HMI tags "2080TN450A01Z02"
   "2080TN450A01Z02.MSW" : 52809b66-421d-457f-8884-6f7a49d4e247 AT %DB5129.DBX18.0, 500 ms
   "2080TN450A01Z02.DefaultText" : TextRef, internal   // Заголовок POPUP окна. При експорте из ECS через скрипт заполняется автоматически, если теги копируются в ручную то требуется в ручную задатать свойство Start Value
   "2080TN450A01Z02.BlockInfo" : Array [0..2] of Int AT %DB5129.DBX38.0, 500 ms
   "2080TN450A01Z02.StatusWork" : Int AT %DB5129.DBW242, 500 ms
   "2080TN450A01Z02.FP_PARAM.DampingTime" : Int AT %DB5129.DBW50, 500 ms
   "2080TN450A01Z02.FP_PARAM.Force_Value" : Real AT %DB5129.DBD52, 500 ms
   "2080TN450A01Z02.FP_PARAM.Scale_Min" : Real AT %DB5129.DBD56, 500 ms
   "2080TN450A01Z02.FP_PARAM.Scale_Max" : Real AT %DB5129.DBD60, 500 ms
   "2080TN450A01Z02.FP_PARAM.Gradient" : Real AT %DB5129.DBD64, 500 ms
   "2080TN450A01Z02.FP_PARAM.Grad_Pos" : Real AT %DB5129.DBD68, 500 ms
   "2080TN450A01Z02.FP_PARAM.Grad_Neg" : Real AT %DB5129.DBD72, 500 ms
   "2080TN450A01Z02.FP_PARAM.Grad_X" : Real AT %DB5129.DBD76, 500 ms
   "2080TN450A01Z02.FP_PARAM.Gradient_Time_Pre" : Int AT %DB5129.DBW80, 500 ms
   "2080TN450A01Z02.FP_PARAM.Gradient_Time_ACC" : Int AT %DB5129.DBW82, 500 ms
   "2080TN450A01Z02.FP_PARAM.Alarm_Hyst" : Real AT %DB5129.DBD84, 500 ms
   "2080TN450A01Z02.FP_PARAM.AlarmLimit_H3" : Real AT %DB5129.DBD88, 500 ms
   "2080TN450A01Z02.FP_PARAM.AlarmLimit_H2" : Real AT %DB5129.DBD92, 500 ms
   "2080TN450A01Z02.FP_PARAM.AlarmLimit_H1" : Real AT %DB5129.DBD96, 500 ms
   "2080TN450A01Z02.FP_PARAM.AlarmLimit_L1" : Real AT %DB5129.DBD100, 500 ms
   "2080TN450A01Z02.FP_PARAM.AlarmLimit_L2" : Real AT %DB5129.DBD104, 500 ms
   "2080TN450A01Z02.FP_PARAM.AlarmLimit_L3" : Real AT %DB5129.DBD108, 500 ms
   "2080TN450A01Z02.FP_PARAM.AlarmDelay_H3_Pre" : Int AT %DB5129.DBW112, 500 ms
   "2080TN450A01Z02.FP_PARAM.AlarmDelay_H3_Acc" : Int AT %DB5129.DBW114, 500 ms
   "2080TN450A01Z02.FP_PARAM.AlarmDelay_H2_Pre" : Int AT %DB5129.DBW116, 500 ms
   "2080TN450A01Z02.FP_PARAM.AlarmDelay_H2_Acc" : Int AT %DB5129.DBW118, 500 ms
   "2080TN450A01Z02.FP_PARAM.AlarmDelay_H1_Pre" : Int AT %DB5129.DBW120, 500 ms
   "2080TN450A01Z02.FP_PARAM.AlarmDelay_H1_Acc" : Int AT %DB5129.DBW122, 500 ms
   "2080TN450A01Z02.FP_PARAM.AlarmDelay_L1_Pre" : Int AT %DB5129.DBW124, 500 ms
   "2080TN450A01Z02.FP_PARAM.AlarmDelay_L1_Acc" : Int AT %DB5129.DBW126, 500 ms
   "2080TN450A01Z02.FP_PARAM.AlarmDelay_L2_Pre" : Int AT %DB5129.DBW128, 500 ms
   "2080TN450A01Z02.FP_PARAM.AlarmDelay_L2_Acc" : Int AT %DB5129.DBW130, 500 ms
   "2080TN450A01Z02.FP_PARAM.AlarmDelay_L3_Pre" : Int AT %DB5129.DBW132, 500 ms
   "2080TN450A01Z02.FP_PARAM.AlarmDelay_L3_Acc" : Int AT %DB5129.DBW134, 500 ms
   "2080TN450A01Z02.FP_PARAM.OpenLoopDelay_Pre" : Int AT %DB5129.DBW136, 500 ms
   "2080TN450A01Z02.FP_PARAM.OpenLoopDelay_Acc" : Int AT %DB5129.DBW138, 500 ms
   "2080TN450A01Z02.FP_PARAM.OverRangeDelay_Pre" : Int AT %DB5129.DBW140, 500 ms
   "2080TN450A01Z02.FP_PARAM.OverRangeDelay_Acc" : Int AT %DB5129.DBW142, 500 ms
   "2080TN450A01Z02.FP_PARAM.AuxLimit_H2_Value" : Real AT %DB5129.DBD144, 500 ms
   "2080TN450A01Z02.FP_PARAM.AuxLimit_H1_Value" : Real AT %DB5129.DBD148, 500 ms
   "2080TN450A01Z02.FP_PARAM.AuxLimit_L2_Value" : Real AT %DB5129.DBD152, 500 ms
   "2080TN450A01Z02.FP_PARAM.AuxLimit_L1_Value" : Real AT %DB5129.DBD156, 500 ms
   "2080TN450A01Z02.Unit" : TextRef, internal   // Еденицы измерения При експорте из ECS через скрипт заполняется автоматически, если теги копируются в ручную то требуется задатать свойство Text
   "2080TN450A01Z02.Decimals" : TextRef, internal   // Формат отображения При експорте из ECS через скрипт, заполняется автоматически. Если теги копируются в ручную то требуется задатать свойство Text s999999.9
   "2080TN450A01Z02.FP_EN.Square" : Bool AT %DB5129.DBX46.0, 500 ms
   "2080TN450A01Z02.FP_EN.SquareRoot" : Bool AT %DB5129.DBX46.1, 500 ms
   "2080TN450A01Z02.FP_EN.ParentSupress" : Bool AT %DB5129.DBX46.2, 500 ms
   "2080TN450A01Z02.FP_EN.ParentSupressUnit" : Bool AT %DB5129.DBX46.3, 500 ms
   "2080TN450A01Z02.FP_EN.Force" : Bool AT %DB5129.DBX46.4, 500 ms
   "2080TN450A01Z02.FP_EN.Damping" : Bool AT %DB5129.DBX46.5, 500 ms
   "2080TN450A01Z02.FP_EN.Gradient_Pos" : Bool AT %DB5129.DBX46.6, 500 ms
   "2080TN450A01Z02.FP_EN.Gradient_Neg" : Bool AT %DB5129.DBX46.7, 500 ms
   "2080TN450A01Z02.FP_EN.Hysteresis" : Bool AT %DB5129.DBX47.0, 500 ms
   "2080TN450A01Z02.FP_EN.Alarm_H3" : Bool AT %DB5129.DBX47.1, 500 ms
   "2080TN450A01Z02.FP_EN.Alarm_H2" : Bool AT %DB5129.DBX47.2, 500 ms
   "2080TN450A01Z02.FP_EN.Alarm_H1" : Bool AT %DB5129.DBX47.3, 500 ms
   "2080TN450A01Z02.FP_EN.Alarm_L1" : Bool AT %DB5129.DBX47.4, 500 ms
   "2080TN450A01Z02.FP_EN.Alarm_L2" : Bool AT %DB5129.DBX47.5, 500 ms
   "2080TN450A01Z02.FP_EN.Alarm_L3" : Bool AT %DB5129.DBX47.6, 500 ms
   "2080TN450A01Z02.FP_EN.AlarmDelay_H3" : Bool AT %DB5129.DBX47.7, 500 ms
   "2080TN450A01Z02.FP_EN.AlarmDelay_H2" : Bool AT %DB5129.DBX48.0, 500 ms
   "2080TN450A01Z02.FP_EN.AlarmDelay_H1" : Bool AT %DB5129.DBX48.1, 500 ms
   "2080TN450A01Z02.FP_EN.AlarmDelay_L1" : Bool AT %DB5129.DBX48.2, 500 ms
   "2080TN450A01Z02.FP_EN.AlarmDelay_L2" : Bool AT %DB5129.DBX48.3, 500 ms
   "2080TN450A01Z02.FP_EN.AlarmDelay_L3" : Bool AT %DB5129.DBX48.4, 500 ms
   "2080TN450A01Z02.FP_EN.ROC_Warn" : Bool AT %DB5129.DBX48.5, 500 ms
   "2080TN450A01Z02.FP_EN.U_Range_Warn" : Bool AT %DB5129.DBX48.6, 500 ms
   "2080TN450A01Z02.FP_EN.O_Range_Warn" : Bool AT %DB5129.DBX48.7, 500 ms
   "2080TN450A01Z02.trend_tag_name" : TextRef, internal   // Еденицы измерения При експорте из ECS через скрипт - заполняется автоматически, если теги копируются в ручную то требуется задатать свойство Text - имя тега для тренда
   "2080TN450A01Z02.DQ.AL_H3" : Bool AT %DB5129.DBX16.0, 500 ms
   "2080TN450A01Z02.DQ.AL_H2" : Bool AT %DB5129.DBX16.1, 500 ms
   "2080TN450A01Z02.DQ.AL_H1" : Bool AT %DB5129.DBX16.2, 500 ms
   "2080TN450A01Z02.DQ.AL_L1" : Bool AT %DB5129.DBX16.3, 500 ms
   "2080TN450A01Z02.DQ.AL_L2" : Bool AT %DB5129.DBX16.4, 500 ms
   "2080TN450A01Z02.DQ.AL_L3" : Bool AT %DB5129.DBX16.5, 500 ms
   "2080TN450A01Z02.DQ.SIG_OK" : Bool AT %DB5129.DBX16.6, 500 ms
   "2080TN450A01Z02.DQ.LIM_H2" : Bool AT %DB5129.DBX16.7, 500 ms
   "2080TN450A01Z02.DQ.LIM_H1" : Bool AT %DB5129.DBX17.0, 500 ms
   "2080TN450A01Z02.DQ.LIM_L1" : Bool AT %DB5129.DBX17.1, 500 ms
   "2080TN450A01Z02.DQ.LIM_L2" : Bool AT %DB5129.DBX17.2, 500 ms
   "2080TN450A01Z02.DQ.GR_P" : Bool AT %DB5129.DBX17.3, 500 ms
   "2080TN450A01Z02.DQ.GR_N" : Bool AT %DB5129.DBX17.4, 500 ms
   "2080TN450A01Z02.I.IN" : Real AT %DB5129.DBD2, 500 ms
   "2080TN450A01Z02.I.SIG_TYPE" : Int AT %DB5129.DBW0, 500 ms
   "2080TN450A01Z02.I.FI_BUS" : Byte AT %DB5129.DBB6, 500 ms
   "2080TN450A01Z02.DI.U_RANGE" : Bool AT %DB5129.DBX7.0, 500 ms
   "2080TN450A01Z02.DI.O_RANGE" : Bool AT %DB5129.DBX7.1, 500 ms
   "2080TN450A01Z02.DI.SIG_FAULT" : Bool AT %DB5129.DBX7.2, 500 ms
   "2080TN450A01Z02.DI.EnConfig" : Bool AT %DB5129.DBX7.3, 500 ms
   "2080TN450A01Z02.DI.AEN" : Bool AT %DB5129.DBX7.4, 500 ms
   "2080TN450A01Z02.DI.AL_SUPR" : Bool AT %DB5129.DBX7.5, 500 ms
   "2080TN450A01Z02.Q.PV_NORM" : Real AT %DB5129.DBD8, 500 ms
   "2080TN450A01Z02.Q.PV_SCAL" : Real AT %DB5129.DBD12, 500 ms
   "2080TN450A01Z02.ParentInfo" : TextRef, internal   // Имя родителя для попап окна, вкладка инфо. При експорте из ECS через скрипт заполняется автоматически, если теги копируются в ручную то требуется в ручную задатать свойство Start Value

HMI tags "2080TN450A01Z03"
   "2080TN450A01Z03.MSW" : 52809b66-421d-457f-8884-6f7a49d4e247 AT %DB5130.DBX18.0, 500 ms
   "2080TN450A01Z03.DefaultText" : TextRef, internal   // Заголовок POPUP окна. При експорте из ECS через скрипт заполняется автоматически, если теги копируются в ручную то требуется в ручную задатать свойство Start Value
   "2080TN450A01Z03.BlockInfo" : Array [0..2] of Int AT %DB5130.DBX38.0, 500 ms
   "2080TN450A01Z03.StatusWork" : Int AT %DB5130.DBW242, 500 ms
   "2080TN450A01Z03.FP_PARAM.DampingTime" : Int AT %DB5130.DBW50, 500 ms
   "2080TN450A01Z03.FP_PARAM.Force_Value" : Real AT %DB5130.DBD52, 500 ms
   "2080TN450A01Z03.FP_PARAM.Scale_Min" : Real AT %DB5130.DBD56, 500 ms
   "2080TN450A01Z03.FP_PARAM.Scale_Max" : Real AT %DB5130.DBD60, 500 ms
   "2080TN450A01Z03.FP_PARAM.Gradient" : Real AT %DB5130.DBD64, 500 ms
   "2080TN450A01Z03.FP_PARAM.Grad_Pos" : Real AT %DB5130.DBD68, 500 ms
   "2080TN450A01Z03.FP_PARAM.Grad_Neg" : Real AT %DB5130.DBD72, 500 ms
   "2080TN450A01Z03.FP_PARAM.Grad_X" : Real AT %DB5130.DBD76, 500 ms
   "2080TN450A01Z03.FP_PARAM.Gradient_Time_Pre" : Int AT %DB5130.DBW80, 500 ms
   "2080TN450A01Z03.FP_PARAM.Gradient_Time_ACC" : Int AT %DB5130.DBW82, 500 ms
   "2080TN450A01Z03.FP_PARAM.Alarm_Hyst" : Real AT %DB5130.DBD84, 500 ms
   "2080TN450A01Z03.FP_PARAM.AlarmLimit_H3" : Real AT %DB5130.DBD88, 500 ms
   "2080TN450A01Z03.FP_PARAM.AlarmLimit_H2" : Real AT %DB5130.DBD92, 500 ms
   "2080TN450A01Z03.FP_PARAM.AlarmLimit_H1" : Real AT %DB5130.DBD96, 500 ms
   "2080TN450A01Z03.FP_PARAM.AlarmLimit_L1" : Real AT %DB5130.DBD100, 500 ms
   "2080TN450A01Z03.FP_PARAM.AlarmLimit_L2" : Real AT %DB5130.DBD104, 500 ms
   "2080TN450A01Z03.FP_PARAM.AlarmLimit_L3" : Real AT %DB5130.DBD108, 500 ms
   "2080TN450A01Z03.FP_PARAM.AlarmDelay_H3_Pre" : Int AT %DB5130.DBW112, 500 ms
   "2080TN450A01Z03.FP_PARAM.AlarmDelay_H3_Acc" : Int AT %DB5130.DBW114, 500 ms
   "2080TN450A01Z03.FP_PARAM.AlarmDelay_H2_Pre" : Int AT %DB5130.DBW116, 500 ms
   "2080TN450A01Z03.FP_PARAM.AlarmDelay_H2_Acc" : Int AT %DB5130.DBW118, 500 ms
   "2080TN450A01Z03.FP_PARAM.AlarmDelay_H1_Pre" : Int AT %DB5130.DBW120, 500 ms
   "2080TN450A01Z03.FP_PARAM.AlarmDelay_H1_Acc" : Int AT %DB5130.DBW122, 500 ms
   "2080TN450A01Z03.FP_PARAM.AlarmDelay_L1_Pre" : Int AT %DB5130.DBW124, 500 ms
   "2080TN450A01Z03.FP_PARAM.AlarmDelay_L1_Acc" : Int AT %DB5130.DBW126, 500 ms
   "2080TN450A01Z03.FP_PARAM.AlarmDelay_L2_Pre" : Int AT %DB5130.DBW128, 500 ms
   "2080TN450A01Z03.FP_PARAM.AlarmDelay_L2_Acc" : Int AT %DB5130.DBW130, 500 ms
   "2080TN450A01Z03.FP_PARAM.AlarmDelay_L3_Pre" : Int AT %DB5130.DBW132, 500 ms
   "2080TN450A01Z03.FP_PARAM.AlarmDelay_L3_Acc" : Int AT %DB5130.DBW134, 500 ms
   "2080TN450A01Z03.FP_PARAM.OpenLoopDelay_Pre" : Int AT %DB5130.DBW136, 500 ms
   "2080TN450A01Z03.FP_PARAM.OpenLoopDelay_Acc" : Int AT %DB5130.DBW138, 500 ms
   "2080TN450A01Z03.FP_PARAM.OverRangeDelay_Pre" : Int AT %DB5130.DBW140, 500 ms
   "2080TN450A01Z03.FP_PARAM.OverRangeDelay_Acc" : Int AT %DB5130.DBW142, 500 ms
   "2080TN450A01Z03.FP_PARAM.AuxLimit_H2_Value" : Real AT %DB5130.DBD144, 500 ms
   "2080TN450A01Z03.FP_PARAM.AuxLimit_H1_Value" : Real AT %DB5130.DBD148, 500 ms
   "2080TN450A01Z03.FP_PARAM.AuxLimit_L2_Value" : Real AT %DB5130.DBD152, 500 ms
   "2080TN450A01Z03.FP_PARAM.AuxLimit_L1_Value" : Real AT %DB5130.DBD156, 500 ms
   "2080TN450A01Z03.Unit" : TextRef, internal   // Еденицы измерения При експорте из ECS через скрипт заполняется автоматически, если теги копируются в ручную то требуется задатать свойство Text
   "2080TN450A01Z03.Decimals" : TextRef, internal   // Формат отображения При експорте из ECS через скрипт, заполняется автоматически. Если теги копируются в ручную то требуется задатать свойство Text s999999.9
   "2080TN450A01Z03.FP_EN.Square" : Bool AT %DB5130.DBX46.0, 500 ms
   "2080TN450A01Z03.FP_EN.SquareRoot" : Bool AT %DB5130.DBX46.1, 500 ms
   "2080TN450A01Z03.FP_EN.ParentSupress" : Bool AT %DB5130.DBX46.2, 500 ms
   "2080TN450A01Z03.FP_EN.ParentSupressUnit" : Bool AT %DB5130.DBX46.3, 500 ms
   "2080TN450A01Z03.FP_EN.Force" : Bool AT %DB5130.DBX46.4, 500 ms
   "2080TN450A01Z03.FP_EN.Damping" : Bool AT %DB5130.DBX46.5, 500 ms
   "2080TN450A01Z03.FP_EN.Gradient_Pos" : Bool AT %DB5130.DBX46.6, 500 ms
   "2080TN450A01Z03.FP_EN.Gradient_Neg" : Bool AT %DB5130.DBX46.7, 500 ms
   "2080TN450A01Z03.FP_EN.Hysteresis" : Bool AT %DB5130.DBX47.0, 500 ms
   "2080TN450A01Z03.FP_EN.Alarm_H3" : Bool AT %DB5130.DBX47.1, 500 ms
   "2080TN450A01Z03.FP_EN.Alarm_H2" : Bool AT %DB5130.DBX47.2, 500 ms
   "2080TN450A01Z03.FP_EN.Alarm_H1" : Bool AT %DB5130.DBX47.3, 500 ms
   "2080TN450A01Z03.FP_EN.Alarm_L1" : Bool AT %DB5130.DBX47.4, 500 ms
   "2080TN450A01Z03.FP_EN.Alarm_L2" : Bool AT %DB5130.DBX47.5, 500 ms
   "2080TN450A01Z03.FP_EN.Alarm_L3" : Bool AT %DB5130.DBX47.6, 500 ms
   "2080TN450A01Z03.FP_EN.AlarmDelay_H3" : Bool AT %DB5130.DBX47.7, 500 ms
   "2080TN450A01Z03.FP_EN.AlarmDelay_H2" : Bool AT %DB5130.DBX48.0, 500 ms
   "2080TN450A01Z03.FP_EN.AlarmDelay_H1" : Bool AT %DB5130.DBX48.1, 500 ms
   "2080TN450A01Z03.FP_EN.AlarmDelay_L1" : Bool AT %DB5130.DBX48.2, 500 ms
   "2080TN450A01Z03.FP_EN.AlarmDelay_L2" : Bool AT %DB5130.DBX48.3, 500 ms
   "2080TN450A01Z03.FP_EN.AlarmDelay_L3" : Bool AT %DB5130.DBX48.4, 500 ms
   "2080TN450A01Z03.FP_EN.ROC_Warn" : Bool AT %DB5130.DBX48.5, 500 ms
   "2080TN450A01Z03.FP_EN.U_Range_Warn" : Bool AT %DB5130.DBX48.6, 500 ms
   "2080TN450A01Z03.FP_EN.O_Range_Warn" : Bool AT %DB5130.DBX48.7, 500 ms
   "2080TN450A01Z03.trend_tag_name" : TextRef, internal   // Еденицы измерения При експорте из ECS через скрипт - заполняется автоматически, если теги копируются в ручную то требуется задатать свойство Text - имя тега для тренда
   "2080TN450A01Z03.DQ.AL_H3" : Bool AT %DB5130.DBX16.0, 500 ms
   "2080TN450A01Z03.DQ.AL_H2" : Bool AT %DB5130.DBX16.1, 500 ms
   "2080TN450A01Z03.DQ.AL_H1" : Bool AT %DB5130.DBX16.2, 500 ms
   "2080TN450A01Z03.DQ.AL_L1" : Bool AT %DB5130.DBX16.3, 500 ms
   "2080TN450A01Z03.DQ.AL_L2" : Bool AT %DB5130.DBX16.4, 500 ms
   "2080TN450A01Z03.DQ.AL_L3" : Bool AT %DB5130.DBX16.5, 500 ms
   "2080TN450A01Z03.DQ.SIG_OK" : Bool AT %DB5130.DBX16.6, 500 ms
   "2080TN450A01Z03.DQ.LIM_H2" : Bool AT %DB5130.DBX16.7, 500 ms
   "2080TN450A01Z03.DQ.LIM_H1" : Bool AT %DB5130.DBX17.0, 500 ms
   "2080TN450A01Z03.DQ.LIM_L1" : Bool AT %DB5130.DBX17.1, 500 ms
   "2080TN450A01Z03.DQ.LIM_L2" : Bool AT %DB5130.DBX17.2, 500 ms
   "2080TN450A01Z03.DQ.GR_P" : Bool AT %DB5130.DBX17.3, 500 ms
   "2080TN450A01Z03.DQ.GR_N" : Bool AT %DB5130.DBX17.4, 500 ms
   "2080TN450A01Z03.I.IN" : Real AT %DB5130.DBD2, 500 ms
   "2080TN450A01Z03.I.SIG_TYPE" : Int AT %DB5130.DBW0, 500 ms
   "2080TN450A01Z03.I.FI_BUS" : Byte AT %DB5130.DBB6, 500 ms
   "2080TN450A01Z03.DI.U_RANGE" : Bool AT %DB5130.DBX7.0, 500 ms
   "2080TN450A01Z03.DI.O_RANGE" : Bool AT %DB5130.DBX7.1, 500 ms
   "2080TN450A01Z03.DI.SIG_FAULT" : Bool AT %DB5130.DBX7.2, 500 ms
   "2080TN450A01Z03.DI.EnConfig" : Bool AT %DB5130.DBX7.3, 500 ms
   "2080TN450A01Z03.DI.AEN" : Bool AT %DB5130.DBX7.4, 500 ms
   "2080TN450A01Z03.DI.AL_SUPR" : Bool AT %DB5130.DBX7.5, 500 ms
   "2080TN450A01Z03.Q.PV_NORM" : Real AT %DB5130.DBD8, 500 ms
   "2080TN450A01Z03.Q.PV_SCAL" : Real AT %DB5130.DBD12, 500 ms
   "2080TN450A01Z03.ParentInfo" : TextRef, internal   // Имя родителя для попап окна, вкладка инфо. При експорте из ECS через скрипт заполняется автоматически, если теги копируются в ручную то требуется в ручную задатать свойство Start Value

HMI tags "2080TN450A01Z05"
   "2080TN450A01Z05.MSW" : 52809b66-421d-457f-8884-6f7a49d4e247 AT %DB5139.DBX18.0, 500 ms
   "2080TN450A01Z05.DefaultText" : TextRef, internal   // Заголовок POPUP окна. При експорте из ECS через скрипт заполняется автоматически, если теги копируются в ручную то требуется в ручную задатать свойство Start Value
   "2080TN450A01Z05.BlockInfo" : Array [0..2] of Int AT %DB5139.DBX38.0, 500 ms
   "2080TN450A01Z05.StatusWork" : Int AT %DB5139.DBW242, 500 ms
   "2080TN450A01Z05.FP_PARAM.DampingTime" : Int AT %DB5139.DBW50, 500 ms
   "2080TN450A01Z05.FP_PARAM.Force_Value" : Real AT %DB5139.DBD52, 500 ms
   "2080TN450A01Z05.FP_PARAM.Scale_Min" : Real AT %DB5139.DBD56, 500 ms
   "2080TN450A01Z05.FP_PARAM.Scale_Max" : Real AT %DB5139.DBD60, 500 ms
   "2080TN450A01Z05.FP_PARAM.Gradient" : Real AT %DB5139.DBD64, 500 ms
   "2080TN450A01Z05.FP_PARAM.Grad_Pos" : Real AT %DB5139.DBD68, 500 ms
   "2080TN450A01Z05.FP_PARAM.Grad_Neg" : Real AT %DB5139.DBD72, 500 ms
   "2080TN450A01Z05.FP_PARAM.Grad_X" : Real AT %DB5139.DBD76, 500 ms
   "2080TN450A01Z05.FP_PARAM.Gradient_Time_Pre" : Int AT %DB5139.DBW80, 500 ms
   "2080TN450A01Z05.FP_PARAM.Gradient_Time_ACC" : Int AT %DB5139.DBW82, 500 ms
   "2080TN450A01Z05.FP_PARAM.Alarm_Hyst" : Real AT %DB5139.DBD84, 500 ms
   "2080TN450A01Z05.FP_PARAM.AlarmLimit_H3" : Real AT %DB5139.DBD88, 500 ms
   "2080TN450A01Z05.FP_PARAM.AlarmLimit_H2" : Real AT %DB5139.DBD92, 500 ms
   "2080TN450A01Z05.FP_PARAM.AlarmLimit_H1" : Real AT %DB5139.DBD96, 500 ms
   "2080TN450A01Z05.FP_PARAM.AlarmLimit_L1" : Real AT %DB5139.DBD100, 500 ms
   "2080TN450A01Z05.FP_PARAM.AlarmLimit_L2" : Real AT %DB5139.DBD104, 500 ms
   "2080TN450A01Z05.FP_PARAM.AlarmLimit_L3" : Real AT %DB5139.DBD108, 500 ms
   "2080TN450A01Z05.FP_PARAM.AlarmDelay_H3_Pre" : Int AT %DB5139.DBW112, 500 ms
   "2080TN450A01Z05.FP_PARAM.AlarmDelay_H3_Acc" : Int AT %DB5139.DBW114, 500 ms
   "2080TN450A01Z05.FP_PARAM.AlarmDelay_H2_Pre" : Int AT %DB5139.DBW116, 500 ms
   "2080TN450A01Z05.FP_PARAM.AlarmDelay_H2_Acc" : Int AT %DB5139.DBW118, 500 ms
   "2080TN450A01Z05.FP_PARAM.AlarmDelay_H1_Pre" : Int AT %DB5139.DBW120, 500 ms
   "2080TN450A01Z05.FP_PARAM.AlarmDelay_H1_Acc" : Int AT %DB5139.DBW122, 500 ms
   "2080TN450A01Z05.FP_PARAM.AlarmDelay_L1_Pre" : Int AT %DB5139.DBW124, 500 ms
   "2080TN450A01Z05.FP_PARAM.AlarmDelay_L1_Acc" : Int AT %DB5139.DBW126, 500 ms
   "2080TN450A01Z05.FP_PARAM.AlarmDelay_L2_Pre" : Int AT %DB5139.DBW128, 500 ms
   "2080TN450A01Z05.FP_PARAM.AlarmDelay_L2_Acc" : Int AT %DB5139.DBW130, 500 ms
   "2080TN450A01Z05.FP_PARAM.AlarmDelay_L3_Pre" : Int AT %DB5139.DBW132, 500 ms
   "2080TN450A01Z05.FP_PARAM.AlarmDelay_L3_Acc" : Int AT %DB5139.DBW134, 500 ms
   "2080TN450A01Z05.FP_PARAM.OpenLoopDelay_Pre" : Int AT %DB5139.DBW136, 500 ms
   "2080TN450A01Z05.FP_PARAM.OpenLoopDelay_Acc" : Int AT %DB5139.DBW138, 500 ms
   "2080TN450A01Z05.FP_PARAM.OverRangeDelay_Pre" : Int AT %DB5139.DBW140, 500 ms
   "2080TN450A01Z05.FP_PARAM.OverRangeDelay_Acc" : Int AT %DB5139.DBW142, 500 ms
   "2080TN450A01Z05.FP_PARAM.AuxLimit_H2_Value" : Real AT %DB5139.DBD144, 500 ms
   "2080TN450A01Z05.FP_PARAM.AuxLimit_H1_Value" : Real AT %DB5139.DBD148, 500 ms
   "2080TN450A01Z05.FP_PARAM.AuxLimit_L2_Value" : Real AT %DB5139.DBD152, 500 ms
   "2080TN450A01Z05.FP_PARAM.AuxLimit_L1_Value" : Real AT %DB5139.DBD156, 500 ms
   "2080TN450A01Z05.Unit" : TextRef, internal   // Еденицы измерения При експорте из ECS через скрипт заполняется автоматически, если теги копируются в ручную то требуется задатать свойство Text
   "2080TN450A01Z05.Decimals" : TextRef, internal   // Формат отображения При експорте из ECS через скрипт, заполняется автоматически. Если теги копируются в ручную то требуется задатать свойство Text s999999.9
   "2080TN450A01Z05.FP_EN.Square" : Bool AT %DB5139.DBX46.0, 500 ms
   "2080TN450A01Z05.FP_EN.SquareRoot" : Bool AT %DB5139.DBX46.1, 500 ms
   "2080TN450A01Z05.FP_EN.ParentSupress" : Bool AT %DB5139.DBX46.2, 500 ms
   "2080TN450A01Z05.FP_EN.ParentSupressUnit" : Bool AT %DB5139.DBX46.3, 500 ms
   "2080TN450A01Z05.FP_EN.Force" : Bool AT %DB5139.DBX46.4, 500 ms
   "2080TN450A01Z05.FP_EN.Damping" : Bool AT %DB5139.DBX46.5, 500 ms
   "2080TN450A01Z05.FP_EN.Gradient_Pos" : Bool AT %DB5139.DBX46.6, 500 ms
   "2080TN450A01Z05.FP_EN.Gradient_Neg" : Bool AT %DB5139.DBX46.7, 500 ms
   "2080TN450A01Z05.FP_EN.Hysteresis" : Bool AT %DB5139.DBX47.0, 500 ms
   "2080TN450A01Z05.FP_EN.Alarm_H3" : Bool AT %DB5139.DBX47.1, 500 ms
   "2080TN450A01Z05.FP_EN.Alarm_H2" : Bool AT %DB5139.DBX47.2, 500 ms
   "2080TN450A01Z05.FP_EN.Alarm_H1" : Bool AT %DB5139.DBX47.3, 500 ms
   "2080TN450A01Z05.FP_EN.Alarm_L1" : Bool AT %DB5139.DBX47.4, 500 ms
   "2080TN450A01Z05.FP_EN.Alarm_L2" : Bool AT %DB5139.DBX47.5, 500 ms
   "2080TN450A01Z05.FP_EN.Alarm_L3" : Bool AT %DB5139.DBX47.6, 500 ms
   "2080TN450A01Z05.FP_EN.AlarmDelay_H3" : Bool AT %DB5139.DBX47.7, 500 ms
   "2080TN450A01Z05.FP_EN.AlarmDelay_H2" : Bool AT %DB5139.DBX48.0, 500 ms
   "2080TN450A01Z05.FP_EN.AlarmDelay_H1" : Bool AT %DB5139.DBX48.1, 500 ms
   "2080TN450A01Z05.FP_EN.AlarmDelay_L1" : Bool AT %DB5139.DBX48.2, 500 ms
   "2080TN450A01Z05.FP_EN.AlarmDelay_L2" : Bool AT %DB5139.DBX48.3, 500 ms
   "2080TN450A01Z05.FP_EN.AlarmDelay_L3" : Bool AT %DB5139.DBX48.4, 500 ms
   "2080TN450A01Z05.FP_EN.ROC_Warn" : Bool AT %DB5139.DBX48.5, 500 ms
   "2080TN450A01Z05.FP_EN.U_Range_Warn" : Bool AT %DB5139.DBX48.6, 500 ms
   "2080TN450A01Z05.FP_EN.O_Range_Warn" : Bool AT %DB5139.DBX48.7, 500 ms
   "2080TN450A01Z05.trend_tag_name" : TextRef, internal   // Еденицы измерения При експорте из ECS через скрипт - заполняется автоматически, если теги копируются в ручную то требуется задатать свойство Text - имя тега для тренда
   "2080TN450A01Z05.DQ.AL_H3" : Bool AT %DB5139.DBX16.0, 500 ms
   "2080TN450A01Z05.DQ.AL_H2" : Bool AT %DB5139.DBX16.1, 500 ms
   "2080TN450A01Z05.DQ.AL_H1" : Bool AT %DB5139.DBX16.2, 500 ms
   "2080TN450A01Z05.DQ.AL_L1" : Bool AT %DB5139.DBX16.3, 500 ms
   "2080TN450A01Z05.DQ.AL_L2" : Bool AT %DB5139.DBX16.4, 500 ms
   "2080TN450A01Z05.DQ.AL_L3" : Bool AT %DB5139.DBX16.5, 500 ms
   "2080TN450A01Z05.DQ.SIG_OK" : Bool AT %DB5139.DBX16.6, 500 ms
   "2080TN450A01Z05.DQ.LIM_H2" : Bool AT %DB5139.DBX16.7, 500 ms
   "2080TN450A01Z05.DQ.LIM_H1" : Bool AT %DB5139.DBX17.0, 500 ms
   "2080TN450A01Z05.DQ.LIM_L1" : Bool AT %DB5139.DBX17.1, 500 ms
   "2080TN450A01Z05.DQ.LIM_L2" : Bool AT %DB5139.DBX17.2, 500 ms
   "2080TN450A01Z05.DQ.GR_P" : Bool AT %DB5139.DBX17.3, 500 ms
   "2080TN450A01Z05.DQ.GR_N" : Bool AT %DB5139.DBX17.4, 500 ms
   "2080TN450A01Z05.I.IN" : Real AT %DB5139.DBD2, 500 ms
   "2080TN450A01Z05.I.SIG_TYPE" : Int AT %DB5139.DBW0, 500 ms
   "2080TN450A01Z05.I.FI_BUS" : Byte AT %DB5139.DBB6, 500 ms
   "2080TN450A01Z05.DI.U_RANGE" : Bool AT %DB5139.DBX7.0, 500 ms
   "2080TN450A01Z05.DI.O_RANGE" : Bool AT %DB5139.DBX7.1, 500 ms
   "2080TN450A01Z05.DI.SIG_FAULT" : Bool AT %DB5139.DBX7.2, 500 ms
   "2080TN450A01Z05.DI.EnConfig" : Bool AT %DB5139.DBX7.3, 500 ms
   "2080TN450A01Z05.DI.AEN" : Bool AT %DB5139.DBX7.4, 500 ms
   "2080TN450A01Z05.DI.AL_SUPR" : Bool AT %DB5139.DBX7.5, 500 ms
   "2080TN450A01Z05.Q.PV_NORM" : Real AT %DB5139.DBD8, 500 ms
   "2080TN450A01Z05.Q.PV_SCAL" : Real AT %DB5139.DBD12, 500 ms
   "2080TN450A01Z05.ParentInfo" : TextRef, internal   // Имя родителя для попап окна, вкладка инфо. При експорте из ECS через скрипт заполняется автоматически, если теги копируются в ручную то требуется в ручную задатать свойство Start Value

HMI tags "2080TN450N01A01"
   "2080TN450N01A01.MSW" : 52809b66-421d-457f-8884-6f7a49d4e247 AT %DB5135.DBX18.0, 500 ms
   "2080TN450N01A01.DefaultText" : TextRef, internal   // Заголовок POPUP окна. При експорте из ECS через скрипт заполняется автоматически, если теги копируются в ручную то требуется в ручную задатать свойство Start Value
   "2080TN450N01A01.BlockInfo" : Array [0..2] of Int AT %DB5135.DBX38.0, 500 ms
   "2080TN450N01A01.StatusWork" : Int AT %DB5135.DBW242, 500 ms
   "2080TN450N01A01.FP_PARAM.DampingTime" : Int AT %DB5135.DBW50, 500 ms
   "2080TN450N01A01.FP_PARAM.Force_Value" : Real AT %DB5135.DBD52, 500 ms
   "2080TN450N01A01.FP_PARAM.Scale_Min" : Real AT %DB5135.DBD56, 500 ms
   "2080TN450N01A01.FP_PARAM.Scale_Max" : Real AT %DB5135.DBD60, 500 ms
   "2080TN450N01A01.FP_PARAM.Gradient" : Real AT %DB5135.DBD64, 500 ms
   "2080TN450N01A01.FP_PARAM.Grad_Pos" : Real AT %DB5135.DBD68, 500 ms
   "2080TN450N01A01.FP_PARAM.Grad_Neg" : Real AT %DB5135.DBD72, 500 ms
   "2080TN450N01A01.FP_PARAM.Grad_X" : Real AT %DB5135.DBD76, 500 ms
   "2080TN450N01A01.FP_PARAM.Gradient_Time_Pre" : Int AT %DB5135.DBW80, 500 ms
   "2080TN450N01A01.FP_PARAM.Gradient_Time_ACC" : Int AT %DB5135.DBW82, 500 ms
   "2080TN450N01A01.FP_PARAM.Alarm_Hyst" : Real AT %DB5135.DBD84, 500 ms
   "2080TN450N01A01.FP_PARAM.AlarmLimit_H3" : Real AT %DB5135.DBD88, 500 ms
   "2080TN450N01A01.FP_PARAM.AlarmLimit_H2" : Real AT %DB5135.DBD92, 500 ms
   "2080TN450N01A01.FP_PARAM.AlarmLimit_H1" : Real AT %DB5135.DBD96, 500 ms
   "2080TN450N01A01.FP_PARAM.AlarmLimit_L1" : Real AT %DB5135.DBD100, 500 ms
   "2080TN450N01A01.FP_PARAM.AlarmLimit_L2" : Real AT %DB5135.DBD104, 500 ms
   "2080TN450N01A01.FP_PARAM.AlarmLimit_L3" : Real AT %DB5135.DBD108, 500 ms
   "2080TN450N01A01.FP_PARAM.AlarmDelay_H3_Pre" : Int AT %DB5135.DBW112, 500 ms
   "2080TN450N01A01.FP_PARAM.AlarmDelay_H3_Acc" : Int AT %DB5135.DBW114, 500 ms
   "2080TN450N01A01.FP_PARAM.AlarmDelay_H2_Pre" : Int AT %DB5135.DBW116, 500 ms
   "2080TN450N01A01.FP_PARAM.AlarmDelay_H2_Acc" : Int AT %DB5135.DBW118, 500 ms
   "2080TN450N01A01.FP_PARAM.AlarmDelay_H1_Pre" : Int AT %DB5135.DBW120, 500 ms
   "2080TN450N01A01.FP_PARAM.AlarmDelay_H1_Acc" : Int AT %DB5135.DBW122, 500 ms
   "2080TN450N01A01.FP_PARAM.AlarmDelay_L1_Pre" : Int AT %DB5135.DBW124, 500 ms
   "2080TN450N01A01.FP_PARAM.AlarmDelay_L1_Acc" : Int AT %DB5135.DBW126, 500 ms
   "2080TN450N01A01.FP_PARAM.AlarmDelay_L2_Pre" : Int AT %DB5135.DBW128, 500 ms
   "2080TN450N01A01.FP_PARAM.AlarmDelay_L2_Acc" : Int AT %DB5135.DBW130, 500 ms
   "2080TN450N01A01.FP_PARAM.AlarmDelay_L3_Pre" : Int AT %DB5135.DBW132, 500 ms
   "2080TN450N01A01.FP_PARAM.AlarmDelay_L3_Acc" : Int AT %DB5135.DBW134, 500 ms
   "2080TN450N01A01.FP_PARAM.OpenLoopDelay_Pre" : Int AT %DB5135.DBW136, 500 ms
   "2080TN450N01A01.FP_PARAM.OpenLoopDelay_Acc" : Int AT %DB5135.DBW138, 500 ms
   "2080TN450N01A01.FP_PARAM.OverRangeDelay_Pre" : Int AT %DB5135.DBW140, 500 ms
   "2080TN450N01A01.FP_PARAM.OverRangeDelay_Acc" : Int AT %DB5135.DBW142, 500 ms
   "2080TN450N01A01.FP_PARAM.AuxLimit_H2_Value" : Real AT %DB5135.DBD144, 500 ms
   "2080TN450N01A01.FP_PARAM.AuxLimit_H1_Value" : Real AT %DB5135.DBD148, 500 ms
   "2080TN450N01A01.FP_PARAM.AuxLimit_L2_Value" : Real AT %DB5135.DBD152, 500 ms
   "2080TN450N01A01.FP_PARAM.AuxLimit_L1_Value" : Real AT %DB5135.DBD156, 500 ms
   "2080TN450N01A01.Unit" : TextRef, internal   // Еденицы измерения При експорте из ECS через скрипт заполняется автоматически, если теги копируются в ручную то требуется задатать свойство Text
   "2080TN450N01A01.Decimals" : TextRef, internal   // Формат отображения При експорте из ECS через скрипт, заполняется автоматически. Если теги копируются в ручную то требуется задатать свойство Text s999999.9
   "2080TN450N01A01.FP_EN.Square" : Bool AT %DB5135.DBX46.0, 500 ms
   "2080TN450N01A01.FP_EN.SquareRoot" : Bool AT %DB5135.DBX46.1, 500 ms
   "2080TN450N01A01.FP_EN.ParentSupress" : Bool AT %DB5135.DBX46.2, 500 ms
   "2080TN450N01A01.FP_EN.ParentSupressUnit" : Bool AT %DB5135.DBX46.3, 500 ms
   "2080TN450N01A01.FP_EN.Force" : Bool AT %DB5135.DBX46.4, 500 ms
   "2080TN450N01A01.FP_EN.Damping" : Bool AT %DB5135.DBX46.5, 500 ms
   "2080TN450N01A01.FP_EN.Gradient_Pos" : Bool AT %DB5135.DBX46.6, 500 ms
   "2080TN450N01A01.FP_EN.Gradient_Neg" : Bool AT %DB5135.DBX46.7, 500 ms
   "2080TN450N01A01.FP_EN.Hysteresis" : Bool AT %DB5135.DBX47.0, 500 ms
   "2080TN450N01A01.FP_EN.Alarm_H3" : Bool AT %DB5135.DBX47.1, 500 ms
   "2080TN450N01A01.FP_EN.Alarm_H2" : Bool AT %DB5135.DBX47.2, 500 ms
   "2080TN450N01A01.FP_EN.Alarm_H1" : Bool AT %DB5135.DBX47.3, 500 ms
   "2080TN450N01A01.FP_EN.Alarm_L1" : Bool AT %DB5135.DBX47.4, 500 ms
   "2080TN450N01A01.FP_EN.Alarm_L2" : Bool AT %DB5135.DBX47.5, 500 ms
   "2080TN450N01A01.FP_EN.Alarm_L3" : Bool AT %DB5135.DBX47.6, 500 ms
   "2080TN450N01A01.FP_EN.AlarmDelay_H3" : Bool AT %DB5135.DBX47.7, 500 ms
   "2080TN450N01A01.FP_EN.AlarmDelay_H2" : Bool AT %DB5135.DBX48.0, 500 ms
   "2080TN450N01A01.FP_EN.AlarmDelay_H1" : Bool AT %DB5135.DBX48.1, 500 ms
   "2080TN450N01A01.FP_EN.AlarmDelay_L1" : Bool AT %DB5135.DBX48.2, 500 ms
   "2080TN450N01A01.FP_EN.AlarmDelay_L2" : Bool AT %DB5135.DBX48.3, 500 ms
   "2080TN450N01A01.FP_EN.AlarmDelay_L3" : Bool AT %DB5135.DBX48.4, 500 ms
   "2080TN450N01A01.FP_EN.ROC_Warn" : Bool AT %DB5135.DBX48.5, 500 ms
   "2080TN450N01A01.FP_EN.U_Range_Warn" : Bool AT %DB5135.DBX48.6, 500 ms
   "2080TN450N01A01.FP_EN.O_Range_Warn" : Bool AT %DB5135.DBX48.7, 500 ms
   "2080TN450N01A01.trend_tag_name" : TextRef, internal   // Еденицы измерения При експорте из ECS через скрипт - заполняется автоматически, если теги копируются в ручную то требуется задатать свойство Text - имя тега для тренда
   "2080TN450N01A01.DQ.AL_H3" : Bool AT %DB5135.DBX16.0, 500 ms
   "2080TN450N01A01.DQ.AL_H2" : Bool AT %DB5135.DBX16.1, 500 ms
   "2080TN450N01A01.DQ.AL_H1" : Bool AT %DB5135.DBX16.2, 500 ms
   "2080TN450N01A01.DQ.AL_L1" : Bool AT %DB5135.DBX16.3, 500 ms
   "2080TN450N01A01.DQ.AL_L2" : Bool AT %DB5135.DBX16.4, 500 ms
   "2080TN450N01A01.DQ.AL_L3" : Bool AT %DB5135.DBX16.5, 500 ms
   "2080TN450N01A01.DQ.SIG_OK" : Bool AT %DB5135.DBX16.6, 500 ms
   "2080TN450N01A01.DQ.LIM_H2" : Bool AT %DB5135.DBX16.7, 500 ms
   "2080TN450N01A01.DQ.LIM_H1" : Bool AT %DB5135.DBX17.0, 500 ms
   "2080TN450N01A01.DQ.LIM_L1" : Bool AT %DB5135.DBX17.1, 500 ms
   "2080TN450N01A01.DQ.LIM_L2" : Bool AT %DB5135.DBX17.2, 500 ms
   "2080TN450N01A01.DQ.GR_P" : Bool AT %DB5135.DBX17.3, 500 ms
   "2080TN450N01A01.DQ.GR_N" : Bool AT %DB5135.DBX17.4, 500 ms
   "2080TN450N01A01.I.IN" : Real AT %DB5135.DBD2, 500 ms
   "2080TN450N01A01.I.SIG_TYPE" : Int AT %DB5135.DBW0, 500 ms
   "2080TN450N01A01.I.FI_BUS" : Byte AT %DB5135.DBB6, 500 ms
   "2080TN450N01A01.DI.U_RANGE" : Bool AT %DB5135.DBX7.0, 500 ms
   "2080TN450N01A01.DI.O_RANGE" : Bool AT %DB5135.DBX7.1, 500 ms
   "2080TN450N01A01.DI.SIG_FAULT" : Bool AT %DB5135.DBX7.2, 500 ms
   "2080TN450N01A01.DI.EnConfig" : Bool AT %DB5135.DBX7.3, 500 ms
   "2080TN450N01A01.DI.AEN" : Bool AT %DB5135.DBX7.4, 500 ms
   "2080TN450N01A01.DI.AL_SUPR" : Bool AT %DB5135.DBX7.5, 500 ms
   "2080TN450N01A01.Q.PV_NORM" : Real AT %DB5135.DBD8, 500 ms
   "2080TN450N01A01.Q.PV_SCAL" : Real AT %DB5135.DBD12, 500 ms
   "2080TN450N01A01.ParentInfo" : TextRef, internal   // Имя родителя для попап окна, вкладка инфо. При експорте из ECS через скрипт заполняется автоматически, если теги копируются в ручную то требуется в ручную задатать свойство Start Value

HMI tags "2080TN450N01I02"
   "2080TN450N01I02.MSW" : 52809b66-421d-457f-8884-6f7a49d4e247 AT %DB5112.DBX18.0, 500 ms
   "2080TN450N01I02.DefaultText" : TextRef, internal   // Заголовок POPUP окна. При експорте из ECS через скрипт заполняется автоматически, если теги копируются в ручную то требуется в ручную задатать свойство Start Value
   "2080TN450N01I02.BlockInfo" : Array [0..2] of Int AT %DB5112.DBX38.0, 500 ms
   "2080TN450N01I02.StatusWork" : Int AT %DB5112.DBW242, 500 ms
   "2080TN450N01I02.FP_PARAM.DampingTime" : Int AT %DB5112.DBW50, 500 ms
   "2080TN450N01I02.FP_PARAM.Force_Value" : Real AT %DB5112.DBD52, 500 ms
   "2080TN450N01I02.FP_PARAM.Scale_Min" : Real AT %DB5112.DBD56, 500 ms
   "2080TN450N01I02.FP_PARAM.Scale_Max" : Real AT %DB5112.DBD60, 500 ms
   "2080TN450N01I02.FP_PARAM.Gradient" : Real AT %DB5112.DBD64, 500 ms
   "2080TN450N01I02.FP_PARAM.Grad_Pos" : Real AT %DB5112.DBD68, 500 ms
   "2080TN450N01I02.FP_PARAM.Grad_Neg" : Real AT %DB5112.DBD72, 500 ms
   "2080TN450N01I02.FP_PARAM.Grad_X" : Real AT %DB5112.DBD76, 500 ms
   "2080TN450N01I02.FP_PARAM.Gradient_Time_Pre" : Int AT %DB5112.DBW80, 500 ms
   "2080TN450N01I02.FP_PARAM.Gradient_Time_ACC" : Int AT %DB5112.DBW82, 500 ms
   "2080TN450N01I02.FP_PARAM.Alarm_Hyst" : Real AT %DB5112.DBD84, 500 ms
   "2080TN450N01I02.FP_PARAM.AlarmLimit_H3" : Real AT %DB5112.DBD88, 500 ms
   "2080TN450N01I02.FP_PARAM.AlarmLimit_H2" : Real AT %DB5112.DBD92, 500 ms
   "2080TN450N01I02.FP_PARAM.AlarmLimit_H1" : Real AT %DB5112.DBD96, 500 ms
   "2080TN450N01I02.FP_PARAM.AlarmLimit_L1" : Real AT %DB5112.DBD100, 500 ms
   "2080TN450N01I02.FP_PARAM.AlarmLimit_L2" : Real AT %DB5112.DBD104, 500 ms
   "2080TN450N01I02.FP_PARAM.AlarmLimit_L3" : Real AT %DB5112.DBD108, 500 ms
   "2080TN450N01I02.FP_PARAM.AlarmDelay_H3_Pre" : Int AT %DB5112.DBW112, 500 ms
   "2080TN450N01I02.FP_PARAM.AlarmDelay_H3_Acc" : Int AT %DB5112.DBW114, 500 ms
   "2080TN450N01I02.FP_PARAM.AlarmDelay_H2_Pre" : Int AT %DB5112.DBW116, 500 ms
   "2080TN450N01I02.FP_PARAM.AlarmDelay_H2_Acc" : Int AT %DB5112.DBW118, 500 ms
   "2080TN450N01I02.FP_PARAM.AlarmDelay_H1_Pre" : Int AT %DB5112.DBW120, 500 ms
   "2080TN450N01I02.FP_PARAM.AlarmDelay_H1_Acc" : Int AT %DB5112.DBW122, 500 ms
   "2080TN450N01I02.FP_PARAM.AlarmDelay_L1_Pre" : Int AT %DB5112.DBW124, 500 ms
   "2080TN450N01I02.FP_PARAM.AlarmDelay_L1_Acc" : Int AT %DB5112.DBW126, 500 ms
   "2080TN450N01I02.FP_PARAM.AlarmDelay_L2_Pre" : Int AT %DB5112.DBW128, 500 ms
   "2080TN450N01I02.FP_PARAM.AlarmDelay_L2_Acc" : Int AT %DB5112.DBW130, 500 ms
   "2080TN450N01I02.FP_PARAM.AlarmDelay_L3_Pre" : Int AT %DB5112.DBW132, 500 ms
   "2080TN450N01I02.FP_PARAM.AlarmDelay_L3_Acc" : Int AT %DB5112.DBW134, 500 ms
   "2080TN450N01I02.FP_PARAM.OpenLoopDelay_Pre" : Int AT %DB5112.DBW136, 500 ms
   "2080TN450N01I02.FP_PARAM.OpenLoopDelay_Acc" : Int AT %DB5112.DBW138, 500 ms
   "2080TN450N01I02.FP_PARAM.OverRangeDelay_Pre" : Int AT %DB5112.DBW140, 500 ms
   "2080TN450N01I02.FP_PARAM.OverRangeDelay_Acc" : Int AT %DB5112.DBW142, 500 ms
   "2080TN450N01I02.FP_PARAM.AuxLimit_H2_Value" : Real AT %DB5112.DBD144, 500 ms
   "2080TN450N01I02.FP_PARAM.AuxLimit_H1_Value" : Real AT %DB5112.DBD148, 500 ms
   "2080TN450N01I02.FP_PARAM.AuxLimit_L2_Value" : Real AT %DB5112.DBD152, 500 ms
   "2080TN450N01I02.FP_PARAM.AuxLimit_L1_Value" : Real AT %DB5112.DBD156, 500 ms
   "2080TN450N01I02.Unit" : TextRef, internal   // Еденицы измерения При експорте из ECS через скрипт заполняется автоматически, если теги копируются в ручную то требуется задатать свойство Text
   "2080TN450N01I02.Decimals" : TextRef, internal   // Формат отображения При експорте из ECS через скрипт, заполняется автоматически. Если теги копируются в ручную то требуется задатать свойство Text s999999.9
   "2080TN450N01I02.FP_EN.Square" : Bool AT %DB5112.DBX46.0, 500 ms
   "2080TN450N01I02.FP_EN.SquareRoot" : Bool AT %DB5112.DBX46.1, 500 ms
   "2080TN450N01I02.FP_EN.ParentSupress" : Bool AT %DB5112.DBX46.2, 500 ms
   "2080TN450N01I02.FP_EN.ParentSupressUnit" : Bool AT %DB5112.DBX46.3, 500 ms
   "2080TN450N01I02.FP_EN.Force" : Bool AT %DB5112.DBX46.4, 500 ms
   "2080TN450N01I02.FP_EN.Damping" : Bool AT %DB5112.DBX46.5, 500 ms
   "2080TN450N01I02.FP_EN.Gradient_Pos" : Bool AT %DB5112.DBX46.6, 500 ms
   "2080TN450N01I02.FP_EN.Gradient_Neg" : Bool AT %DB5112.DBX46.7, 500 ms
   "2080TN450N01I02.FP_EN.Hysteresis" : Bool AT %DB5112.DBX47.0, 500 ms
   "2080TN450N01I02.FP_EN.Alarm_H3" : Bool AT %DB5112.DBX47.1, 500 ms
   "2080TN450N01I02.FP_EN.Alarm_H2" : Bool AT %DB5112.DBX47.2, 500 ms
   "2080TN450N01I02.FP_EN.Alarm_H1" : Bool AT %DB5112.DBX47.3, 500 ms
   "2080TN450N01I02.FP_EN.Alarm_L1" : Bool AT %DB5112.DBX47.4, 500 ms
   "2080TN450N01I02.FP_EN.Alarm_L2" : Bool AT %DB5112.DBX47.5, 500 ms
   "2080TN450N01I02.FP_EN.Alarm_L3" : Bool AT %DB5112.DBX47.6, 500 ms
   "2080TN450N01I02.FP_EN.AlarmDelay_H3" : Bool AT %DB5112.DBX47.7, 500 ms
   "2080TN450N01I02.FP_EN.AlarmDelay_H2" : Bool AT %DB5112.DBX48.0, 500 ms
   "2080TN450N01I02.FP_EN.AlarmDelay_H1" : Bool AT %DB5112.DBX48.1, 500 ms
   "2080TN450N01I02.FP_EN.AlarmDelay_L1" : Bool AT %DB5112.DBX48.2, 500 ms
   "2080TN450N01I02.FP_EN.AlarmDelay_L2" : Bool AT %DB5112.DBX48.3, 500 ms
   "2080TN450N01I02.FP_EN.AlarmDelay_L3" : Bool AT %DB5112.DBX48.4, 500 ms
   "2080TN450N01I02.FP_EN.ROC_Warn" : Bool AT %DB5112.DBX48.5, 500 ms
   "2080TN450N01I02.FP_EN.U_Range_Warn" : Bool AT %DB5112.DBX48.6, 500 ms
   "2080TN450N01I02.FP_EN.O_Range_Warn" : Bool AT %DB5112.DBX48.7, 500 ms
   "2080TN450N01I02.trend_tag_name" : TextRef, internal   // Еденицы измерения При експорте из ECS через скрипт - заполняется автоматически, если теги копируются в ручную то требуется задатать свойство Text - имя тега для тренда
   "2080TN450N01I02.DQ.AL_H3" : Bool AT %DB5112.DBX16.0, 500 ms
   "2080TN450N01I02.DQ.AL_H2" : Bool AT %DB5112.DBX16.1, 500 ms
   "2080TN450N01I02.DQ.AL_H1" : Bool AT %DB5112.DBX16.2, 500 ms
   "2080TN450N01I02.DQ.AL_L1" : Bool AT %DB5112.DBX16.3, 500 ms
   "2080TN450N01I02.DQ.AL_L2" : Bool AT %DB5112.DBX16.4, 500 ms
   "2080TN450N01I02.DQ.AL_L3" : Bool AT %DB5112.DBX16.5, 500 ms
   "2080TN450N01I02.DQ.SIG_OK" : Bool AT %DB5112.DBX16.6, 500 ms
   "2080TN450N01I02.DQ.LIM_H2" : Bool AT %DB5112.DBX16.7, 500 ms
   "2080TN450N01I02.DQ.LIM_H1" : Bool AT %DB5112.DBX17.0, 500 ms
   "2080TN450N01I02.DQ.LIM_L1" : Bool AT %DB5112.DBX17.1, 500 ms
   "2080TN450N01I02.DQ.LIM_L2" : Bool AT %DB5112.DBX17.2, 500 ms
   "2080TN450N01I02.DQ.GR_P" : Bool AT %DB5112.DBX17.3, 500 ms
   "2080TN450N01I02.DQ.GR_N" : Bool AT %DB5112.DBX17.4, 500 ms
   "2080TN450N01I02.I.IN" : Real AT %DB5112.DBD2, 500 ms
   "2080TN450N01I02.I.SIG_TYPE" : Int AT %DB5112.DBW0, 500 ms
   "2080TN450N01I02.I.FI_BUS" : Byte AT %DB5112.DBB6, 500 ms
   "2080TN450N01I02.DI.U_RANGE" : Bool AT %DB5112.DBX7.0, 500 ms
   "2080TN450N01I02.DI.O_RANGE" : Bool AT %DB5112.DBX7.1, 500 ms
   "2080TN450N01I02.DI.SIG_FAULT" : Bool AT %DB5112.DBX7.2, 500 ms
   "2080TN450N01I02.DI.EnConfig" : Bool AT %DB5112.DBX7.3, 500 ms
   "2080TN450N01I02.DI.AEN" : Bool AT %DB5112.DBX7.4, 500 ms
   "2080TN450N01I02.DI.AL_SUPR" : Bool AT %DB5112.DBX7.5, 500 ms
   "2080TN450N01I02.Q.PV_NORM" : Real AT %DB5112.DBD8, 500 ms
   "2080TN450N01I02.Q.PV_SCAL" : Real AT %DB5112.DBD12, 500 ms
   "2080TN450N01I02.ParentInfo" : TextRef, internal   // Имя родителя для попап окна, вкладка инфо. При експорте из ECS через скрипт заполняется автоматически, если теги копируются в ручную то требуется в ручную задатать свойство Start Value

HMI tags "2080TN450N01I04"
   "2080TN450N01I04.MSW" : 52809b66-421d-457f-8884-6f7a49d4e247 AT %DB5113.DBX18.0, 500 ms
   "2080TN450N01I04.DefaultText" : TextRef, internal   // Заголовок POPUP окна. При експорте из ECS через скрипт заполняется автоматически, если теги копируются в ручную то требуется в ручную задатать свойство Start Value
   "2080TN450N01I04.BlockInfo" : Array [0..2] of Int AT %DB5113.DBX38.0, 500 ms
   "2080TN450N01I04.StatusWork" : Int AT %DB5113.DBW242, 500 ms
   "2080TN450N01I04.FP_PARAM.DampingTime" : Int AT %DB5113.DBW50, 500 ms
   "2080TN450N01I04.FP_PARAM.Force_Value" : Real AT %DB5113.DBD52, 500 ms
   "2080TN450N01I04.FP_PARAM.Scale_Min" : Real AT %DB5113.DBD56, 500 ms
   "2080TN450N01I04.FP_PARAM.Scale_Max" : Real AT %DB5113.DBD60, 500 ms
   "2080TN450N01I04.FP_PARAM.Gradient" : Real AT %DB5113.DBD64, 500 ms
   "2080TN450N01I04.FP_PARAM.Grad_Pos" : Real AT %DB5113.DBD68, 500 ms
   "2080TN450N01I04.FP_PARAM.Grad_Neg" : Real AT %DB5113.DBD72, 500 ms
   "2080TN450N01I04.FP_PARAM.Grad_X" : Real AT %DB5113.DBD76, 500 ms
   "2080TN450N01I04.FP_PARAM.Gradient_Time_Pre" : Int AT %DB5113.DBW80, 500 ms
   "2080TN450N01I04.FP_PARAM.Gradient_Time_ACC" : Int AT %DB5113.DBW82, 500 ms
   "2080TN450N01I04.FP_PARAM.Alarm_Hyst" : Real AT %DB5113.DBD84, 500 ms
   "2080TN450N01I04.FP_PARAM.AlarmLimit_H3" : Real AT %DB5113.DBD88, 500 ms
   "2080TN450N01I04.FP_PARAM.AlarmLimit_H2" : Real AT %DB5113.DBD92, 500 ms
   "2080TN450N01I04.FP_PARAM.AlarmLimit_H1" : Real AT %DB5113.DBD96, 500 ms
   "2080TN450N01I04.FP_PARAM.AlarmLimit_L1" : Real AT %DB5113.DBD100, 500 ms
   "2080TN450N01I04.FP_PARAM.AlarmLimit_L2" : Real AT %DB5113.DBD104, 500 ms
   "2080TN450N01I04.FP_PARAM.AlarmLimit_L3" : Real AT %DB5113.DBD108, 500 ms
   "2080TN450N01I04.FP_PARAM.AlarmDelay_H3_Pre" : Int AT %DB5113.DBW112, 500 ms
   "2080TN450N01I04.FP_PARAM.AlarmDelay_H3_Acc" : Int AT %DB5113.DBW114, 500 ms
   "2080TN450N01I04.FP_PARAM.AlarmDelay_H2_Pre" : Int AT %DB5113.DBW116, 500 ms
   "2080TN450N01I04.FP_PARAM.AlarmDelay_H2_Acc" : Int AT %DB5113.DBW118, 500 ms
   "2080TN450N01I04.FP_PARAM.AlarmDelay_H1_Pre" : Int AT %DB5113.DBW120, 500 ms
   "2080TN450N01I04.FP_PARAM.AlarmDelay_H1_Acc" : Int AT %DB5113.DBW122, 500 ms
   "2080TN450N01I04.FP_PARAM.AlarmDelay_L1_Pre" : Int AT %DB5113.DBW124, 500 ms
   "2080TN450N01I04.FP_PARAM.AlarmDelay_L1_Acc" : Int AT %DB5113.DBW126, 500 ms
   "2080TN450N01I04.FP_PARAM.AlarmDelay_L2_Pre" : Int AT %DB5113.DBW128, 500 ms
   "2080TN450N01I04.FP_PARAM.AlarmDelay_L2_Acc" : Int AT %DB5113.DBW130, 500 ms
   "2080TN450N01I04.FP_PARAM.AlarmDelay_L3_Pre" : Int AT %DB5113.DBW132, 500 ms
   "2080TN450N01I04.FP_PARAM.AlarmDelay_L3_Acc" : Int AT %DB5113.DBW134, 500 ms
   "2080TN450N01I04.FP_PARAM.OpenLoopDelay_Pre" : Int AT %DB5113.DBW136, 500 ms
   "2080TN450N01I04.FP_PARAM.OpenLoopDelay_Acc" : Int AT %DB5113.DBW138, 500 ms
   "2080TN450N01I04.FP_PARAM.OverRangeDelay_Pre" : Int AT %DB5113.DBW140, 500 ms
   "2080TN450N01I04.FP_PARAM.OverRangeDelay_Acc" : Int AT %DB5113.DBW142, 500 ms
   "2080TN450N01I04.FP_PARAM.AuxLimit_H2_Value" : Real AT %DB5113.DBD144, 500 ms
   "2080TN450N01I04.FP_PARAM.AuxLimit_H1_Value" : Real AT %DB5113.DBD148, 500 ms
   "2080TN450N01I04.FP_PARAM.AuxLimit_L2_Value" : Real AT %DB5113.DBD152, 500 ms
   "2080TN450N01I04.FP_PARAM.AuxLimit_L1_Value" : Real AT %DB5113.DBD156, 500 ms
   "2080TN450N01I04.Unit" : TextRef, internal   // Еденицы измерения При експорте из ECS через скрипт заполняется автоматически, если теги копируются в ручную то требуется задатать свойство Text
   "2080TN450N01I04.Decimals" : TextRef, internal   // Формат отображения При експорте из ECS через скрипт, заполняется автоматически. Если теги копируются в ручную то требуется задатать свойство Text s999999.9
   "2080TN450N01I04.FP_EN.Square" : Bool AT %DB5113.DBX46.0, 500 ms
   "2080TN450N01I04.FP_EN.SquareRoot" : Bool AT %DB5113.DBX46.1, 500 ms
   "2080TN450N01I04.FP_EN.ParentSupress" : Bool AT %DB5113.DBX46.2, 500 ms
   "2080TN450N01I04.FP_EN.ParentSupressUnit" : Bool AT %DB5113.DBX46.3, 500 ms
   "2080TN450N01I04.FP_EN.Force" : Bool AT %DB5113.DBX46.4, 500 ms
   "2080TN450N01I04.FP_EN.Damping" : Bool AT %DB5113.DBX46.5, 500 ms
   "2080TN450N01I04.FP_EN.Gradient_Pos" : Bool AT %DB5113.DBX46.6, 500 ms
   "2080TN450N01I04.FP_EN.Gradient_Neg" : Bool AT %DB5113.DBX46.7, 500 ms
   "2080TN450N01I04.FP_EN.Hysteresis" : Bool AT %DB5113.DBX47.0, 500 ms
   "2080TN450N01I04.FP_EN.Alarm_H3" : Bool AT %DB5113.DBX47.1, 500 ms
   "2080TN450N01I04.FP_EN.Alarm_H2" : Bool AT %DB5113.DBX47.2, 500 ms
   "2080TN450N01I04.FP_EN.Alarm_H1" : Bool AT %DB5113.DBX47.3, 500 ms
   "2080TN450N01I04.FP_EN.Alarm_L1" : Bool AT %DB5113.DBX47.4, 500 ms
   "2080TN450N01I04.FP_EN.Alarm_L2" : Bool AT %DB5113.DBX47.5, 500 ms
   "2080TN450N01I04.FP_EN.Alarm_L3" : Bool AT %DB5113.DBX47.6, 500 ms
   "2080TN450N01I04.FP_EN.AlarmDelay_H3" : Bool AT %DB5113.DBX47.7, 500 ms
   "2080TN450N01I04.FP_EN.AlarmDelay_H2" : Bool AT %DB5113.DBX48.0, 500 ms
   "2080TN450N01I04.FP_EN.AlarmDelay_H1" : Bool AT %DB5113.DBX48.1, 500 ms
   "2080TN450N01I04.FP_EN.AlarmDelay_L1" : Bool AT %DB5113.DBX48.2, 500 ms
   "2080TN450N01I04.FP_EN.AlarmDelay_L2" : Bool AT %DB5113.DBX48.3, 500 ms
   "2080TN450N01I04.FP_EN.AlarmDelay_L3" : Bool AT %DB5113.DBX48.4, 500 ms
   "2080TN450N01I04.FP_EN.ROC_Warn" : Bool AT %DB5113.DBX48.5, 500 ms
   "2080TN450N01I04.FP_EN.U_Range_Warn" : Bool AT %DB5113.DBX48.6, 500 ms
   "2080TN450N01I04.FP_EN.O_Range_Warn" : Bool AT %DB5113.DBX48.7, 500 ms
   "2080TN450N01I04.trend_tag_name" : TextRef, internal   // Еденицы измерения При експорте из ECS через скрипт - заполняется автоматически, если теги копируются в ручную то требуется задатать свойство Text - имя тега для тренда
   "2080TN450N01I04.DQ.AL_H3" : Bool AT %DB5113.DBX16.0, 500 ms
   "2080TN450N01I04.DQ.AL_H2" : Bool AT %DB5113.DBX16.1, 500 ms
   "2080TN450N01I04.DQ.AL_H1" : Bool AT %DB5113.DBX16.2, 500 ms
   "2080TN450N01I04.DQ.AL_L1" : Bool AT %DB5113.DBX16.3, 500 ms
   "2080TN450N01I04.DQ.AL_L2" : Bool AT %DB5113.DBX16.4, 500 ms
   "2080TN450N01I04.DQ.AL_L3" : Bool AT %DB5113.DBX16.5, 500 ms
   "2080TN450N01I04.DQ.SIG_OK" : Bool AT %DB5113.DBX16.6, 500 ms
   "2080TN450N01I04.DQ.LIM_H2" : Bool AT %DB5113.DBX16.7, 500 ms
   "2080TN450N01I04.DQ.LIM_H1" : Bool AT %DB5113.DBX17.0, 500 ms
   "2080TN450N01I04.DQ.LIM_L1" : Bool AT %DB5113.DBX17.1, 500 ms
   "2080TN450N01I04.DQ.LIM_L2" : Bool AT %DB5113.DBX17.2, 500 ms
   "2080TN450N01I04.DQ.GR_P" : Bool AT %DB5113.DBX17.3, 500 ms
   "2080TN450N01I04.DQ.GR_N" : Bool AT %DB5113.DBX17.4, 500 ms
   "2080TN450N01I04.I.IN" : Real AT %DB5113.DBD2, 500 ms
   "2080TN450N01I04.I.SIG_TYPE" : Int AT %DB5113.DBW0, 500 ms
   "2080TN450N01I04.I.FI_BUS" : Byte AT %DB5113.DBB6, 500 ms
   "2080TN450N01I04.DI.U_RANGE" : Bool AT %DB5113.DBX7.0, 500 ms
   "2080TN450N01I04.DI.O_RANGE" : Bool AT %DB5113.DBX7.1, 500 ms
   "2080TN450N01I04.DI.SIG_FAULT" : Bool AT %DB5113.DBX7.2, 500 ms
   "2080TN450N01I04.DI.EnConfig" : Bool AT %DB5113.DBX7.3, 500 ms
   "2080TN450N01I04.DI.AEN" : Bool AT %DB5113.DBX7.4, 500 ms
   "2080TN450N01I04.DI.AL_SUPR" : Bool AT %DB5113.DBX7.5, 500 ms
   "2080TN450N01I04.Q.PV_NORM" : Real AT %DB5113.DBD8, 500 ms
   "2080TN450N01I04.Q.PV_SCAL" : Real AT %DB5113.DBD12, 500 ms
   "2080TN450N01I04.ParentInfo" : TextRef, internal   // Имя родителя для попап окна, вкладка инфо. При експорте из ECS через скрипт заполняется автоматически, если теги копируются в ручную то требуется в ручную задатать свойство Start Value

HMI tags "2080TN450N02P01"
   "2080TN450N02P01.MSW" : 52809b66-421d-457f-8884-6f7a49d4e247 AT %DB5136.DBX18.0, 500 ms
   "2080TN450N02P01.DefaultText" : TextRef, internal   // Заголовок POPUP окна. При експорте из ECS через скрипт заполняется автоматически, если теги копируются в ручную то требуется в ручную задатать свойство Start Value
   "2080TN450N02P01.BlockInfo" : Array [0..2] of Int AT %DB5136.DBX38.0, 500 ms
   "2080TN450N02P01.StatusWork" : Int AT %DB5136.DBW242, 500 ms
   "2080TN450N02P01.FP_PARAM.DampingTime" : Int AT %DB5136.DBW50, 500 ms
   "2080TN450N02P01.FP_PARAM.Force_Value" : Real AT %DB5136.DBD52, 500 ms
   "2080TN450N02P01.FP_PARAM.Scale_Min" : Real AT %DB5136.DBD56, 500 ms
   "2080TN450N02P01.FP_PARAM.Scale_Max" : Real AT %DB5136.DBD60, 500 ms
   "2080TN450N02P01.FP_PARAM.Gradient" : Real AT %DB5136.DBD64, 500 ms
   "2080TN450N02P01.FP_PARAM.Grad_Pos" : Real AT %DB5136.DBD68, 500 ms
   "2080TN450N02P01.FP_PARAM.Grad_Neg" : Real AT %DB5136.DBD72, 500 ms
   "2080TN450N02P01.FP_PARAM.Grad_X" : Real AT %DB5136.DBD76, 500 ms
   "2080TN450N02P01.FP_PARAM.Gradient_Time_Pre" : Int AT %DB5136.DBW80, 500 ms
   "2080TN450N02P01.FP_PARAM.Gradient_Time_ACC" : Int AT %DB5136.DBW82, 500 ms
   "2080TN450N02P01.FP_PARAM.Alarm_Hyst" : Real AT %DB5136.DBD84, 500 ms
   "2080TN450N02P01.FP_PARAM.AlarmLimit_H3" : Real AT %DB5136.DBD88, 500 ms
   "2080TN450N02P01.FP_PARAM.AlarmLimit_H2" : Real AT %DB5136.DBD92, 500 ms
   "2080TN450N02P01.FP_PARAM.AlarmLimit_H1" : Real AT %DB5136.DBD96, 500 ms
   "2080TN450N02P01.FP_PARAM.AlarmLimit_L1" : Real AT %DB5136.DBD100, 500 ms
   "2080TN450N02P01.FP_PARAM.AlarmLimit_L2" : Real AT %DB5136.DBD104, 500 ms
   "2080TN450N02P01.FP_PARAM.AlarmLimit_L3" : Real AT %DB5136.DBD108, 500 ms
   "2080TN450N02P01.FP_PARAM.AlarmDelay_H3_Pre" : Int AT %DB5136.DBW112, 500 ms
   "2080TN450N02P01.FP_PARAM.AlarmDelay_H3_Acc" : Int AT %DB5136.DBW114, 500 ms
   "2080TN450N02P01.FP_PARAM.AlarmDelay_H2_Pre" : Int AT %DB5136.DBW116, 500 ms
   "2080TN450N02P01.FP_PARAM.AlarmDelay_H2_Acc" : Int AT %DB5136.DBW118, 500 ms
   "2080TN450N02P01.FP_PARAM.AlarmDelay_H1_Pre" : Int AT %DB5136.DBW120, 500 ms
   "2080TN450N02P01.FP_PARAM.AlarmDelay_H1_Acc" : Int AT %DB5136.DBW122, 500 ms
   "2080TN450N02P01.FP_PARAM.AlarmDelay_L1_Pre" : Int AT %DB5136.DBW124, 500 ms
   "2080TN450N02P01.FP_PARAM.AlarmDelay_L1_Acc" : Int AT %DB5136.DBW126, 500 ms
   "2080TN450N02P01.FP_PARAM.AlarmDelay_L2_Pre" : Int AT %DB5136.DBW128, 500 ms
   "2080TN450N02P01.FP_PARAM.AlarmDelay_L2_Acc" : Int AT %DB5136.DBW130, 500 ms
   "2080TN450N02P01.FP_PARAM.AlarmDelay_L3_Pre" : Int AT %DB5136.DBW132, 500 ms
   "2080TN450N02P01.FP_PARAM.AlarmDelay_L3_Acc" : Int AT %DB5136.DBW134, 500 ms
   "2080TN450N02P01.FP_PARAM.OpenLoopDelay_Pre" : Int AT %DB5136.DBW136, 500 ms
   "2080TN450N02P01.FP_PARAM.OpenLoopDelay_Acc" : Int AT %DB5136.DBW138, 500 ms
   "2080TN450N02P01.FP_PARAM.OverRangeDelay_Pre" : Int AT %DB5136.DBW140, 500 ms
   "2080TN450N02P01.FP_PARAM.OverRangeDelay_Acc" : Int AT %DB5136.DBW142, 500 ms
   "2080TN450N02P01.FP_PARAM.AuxLimit_H2_Value" : Real AT %DB5136.DBD144, 500 ms
   "2080TN450N02P01.FP_PARAM.AuxLimit_H1_Value" : Real AT %DB5136.DBD148, 500 ms
   "2080TN450N02P01.FP_PARAM.AuxLimit_L2_Value" : Real AT %DB5136.DBD152, 500 ms
   "2080TN450N02P01.FP_PARAM.AuxLimit_L1_Value" : Real AT %DB5136.DBD156, 500 ms
   "2080TN450N02P01.Unit" : TextRef, internal   // Еденицы измерения При експорте из ECS через скрипт заполняется автоматически, если теги копируются в ручную то требуется задатать свойство Text
   "2080TN450N02P01.Decimals" : TextRef, internal   // Формат отображения При експорте из ECS через скрипт, заполняется автоматически. Если теги копируются в ручную то требуется задатать свойство Text s999999.9
   "2080TN450N02P01.FP_EN.Square" : Bool AT %DB5136.DBX46.0, 500 ms
   "2080TN450N02P01.FP_EN.SquareRoot" : Bool AT %DB5136.DBX46.1, 500 ms
   "2080TN450N02P01.FP_EN.ParentSupress" : Bool AT %DB5136.DBX46.2, 500 ms
   "2080TN450N02P01.FP_EN.ParentSupressUnit" : Bool AT %DB5136.DBX46.3, 500 ms
   "2080TN450N02P01.FP_EN.Force" : Bool AT %DB5136.DBX46.4, 500 ms
   "2080TN450N02P01.FP_EN.Damping" : Bool AT %DB5136.DBX46.5, 500 ms
   "2080TN450N02P01.FP_EN.Gradient_Pos" : Bool AT %DB5136.DBX46.6, 500 ms
   "2080TN450N02P01.FP_EN.Gradient_Neg" : Bool AT %DB5136.DBX46.7, 500 ms
   "2080TN450N02P01.FP_EN.Hysteresis" : Bool AT %DB5136.DBX47.0, 500 ms
   "2080TN450N02P01.FP_EN.Alarm_H3" : Bool AT %DB5136.DBX47.1, 500 ms
   "2080TN450N02P01.FP_EN.Alarm_H2" : Bool AT %DB5136.DBX47.2, 500 ms
   "2080TN450N02P01.FP_EN.Alarm_H1" : Bool AT %DB5136.DBX47.3, 500 ms
   "2080TN450N02P01.FP_EN.Alarm_L1" : Bool AT %DB5136.DBX47.4, 500 ms
   "2080TN450N02P01.FP_EN.Alarm_L2" : Bool AT %DB5136.DBX47.5, 500 ms
   "2080TN450N02P01.FP_EN.Alarm_L3" : Bool AT %DB5136.DBX47.6, 500 ms
   "2080TN450N02P01.FP_EN.AlarmDelay_H3" : Bool AT %DB5136.DBX47.7, 500 ms
   "2080TN450N02P01.FP_EN.AlarmDelay_H2" : Bool AT %DB5136.DBX48.0, 500 ms
   "2080TN450N02P01.FP_EN.AlarmDelay_H1" : Bool AT %DB5136.DBX48.1, 500 ms
   "2080TN450N02P01.FP_EN.AlarmDelay_L1" : Bool AT %DB5136.DBX48.2, 500 ms
   "2080TN450N02P01.FP_EN.AlarmDelay_L2" : Bool AT %DB5136.DBX48.3, 500 ms
   "2080TN450N02P01.FP_EN.AlarmDelay_L3" : Bool AT %DB5136.DBX48.4, 500 ms
   "2080TN450N02P01.FP_EN.ROC_Warn" : Bool AT %DB5136.DBX48.5, 500 ms
   "2080TN450N02P01.FP_EN.U_Range_Warn" : Bool AT %DB5136.DBX48.6, 500 ms
   "2080TN450N02P01.FP_EN.O_Range_Warn" : Bool AT %DB5136.DBX48.7, 500 ms
   "2080TN450N02P01.trend_tag_name" : TextRef, internal   // Еденицы измерения При експорте из ECS через скрипт - заполняется автоматически, если теги копируются в ручную то требуется задатать свойство Text - имя тега для тренда
   "2080TN450N02P01.DQ.AL_H3" : Bool AT %DB5136.DBX16.0, 500 ms
   "2080TN450N02P01.DQ.AL_H2" : Bool AT %DB5136.DBX16.1, 500 ms
   "2080TN450N02P01.DQ.AL_H1" : Bool AT %DB5136.DBX16.2, 500 ms
   "2080TN450N02P01.DQ.AL_L1" : Bool AT %DB5136.DBX16.3, 500 ms
   "2080TN450N02P01.DQ.AL_L2" : Bool AT %DB5136.DBX16.4, 500 ms
   "2080TN450N02P01.DQ.AL_L3" : Bool AT %DB5136.DBX16.5, 500 ms
   "2080TN450N02P01.DQ.SIG_OK" : Bool AT %DB5136.DBX16.6, 500 ms
   "2080TN450N02P01.DQ.LIM_H2" : Bool AT %DB5136.DBX16.7, 500 ms
   "2080TN450N02P01.DQ.LIM_H1" : Bool AT %DB5136.DBX17.0, 500 ms
   "2080TN450N02P01.DQ.LIM_L1" : Bool AT %DB5136.DBX17.1, 500 ms
   "2080TN450N02P01.DQ.LIM_L2" : Bool AT %DB5136.DBX17.2, 500 ms
   "2080TN450N02P01.DQ.GR_P" : Bool AT %DB5136.DBX17.3, 500 ms
   "2080TN450N02P01.DQ.GR_N" : Bool AT %DB5136.DBX17.4, 500 ms
   "2080TN450N02P01.I.IN" : Real AT %DB5136.DBD2, 500 ms
   "2080TN450N02P01.I.SIG_TYPE" : Int AT %DB5136.DBW0, 500 ms
   "2080TN450N02P01.I.FI_BUS" : Byte AT %DB5136.DBB6, 500 ms
   "2080TN450N02P01.DI.U_RANGE" : Bool AT %DB5136.DBX7.0, 500 ms
   "2080TN450N02P01.DI.O_RANGE" : Bool AT %DB5136.DBX7.1, 500 ms
   "2080TN450N02P01.DI.SIG_FAULT" : Bool AT %DB5136.DBX7.2, 500 ms
   "2080TN450N02P01.DI.EnConfig" : Bool AT %DB5136.DBX7.3, 500 ms
   "2080TN450N02P01.DI.AEN" : Bool AT %DB5136.DBX7.4, 500 ms
   "2080TN450N02P01.DI.AL_SUPR" : Bool AT %DB5136.DBX7.5, 500 ms
   "2080TN450N02P01.Q.PV_NORM" : Real AT %DB5136.DBD8, 500 ms
   "2080TN450N02P01.Q.PV_SCAL" : Real AT %DB5136.DBD12, 500 ms
   "2080TN450N02P01.ParentInfo" : TextRef, internal   // Имя родителя для попап окна, вкладка инфо. При експорте из ECS через скрипт заполняется автоматически, если теги копируются в ручную то требуется в ручную задатать свойство Start Value

HMI tags "2080SP241Y01"
   "2080SP241Y01.DefaultText" : TextRef, internal   // Заголовок POPUP окна. При експорте из ECS через скрипт заполняется автоматически, если теги копируются в ручную то требуется в ручную задатать свойство Start Value
   "2080SP241Y01.StatusWork" : Int AT %DB4330.DBW458, 500 ms
   "2080SP241Y01.ModePointer" : Int AT %DB4330.DBW460, 500 ms
   "2080SP241Y01.FP_CMD.Start1" : Bool AT %DB4330.DBX79.3, 500 ms
   "2080SP241Y01.FP_CMD.Start2" : Bool AT %DB4330.DBX79.4, 500 ms
   "2080SP241Y01.FP_CMD.Stop" : Bool AT %DB4330.DBX79.6, 500 ms
   "2080SP241Y01.FP_CMD.AckAlarm" : Bool AT %DB4330.DBX78.7, 500 ms
   "2080SP241Y01.FP_CMD.Auto" : Bool AT %DB4330.DBX79.0, 500 ms
   "2080SP241Y01.FP_CMD.Local" : Bool AT %DB4330.DBX79.2, 500 ms
   "2080SP241Y01.FP_CMD.Manual" : Bool AT %DB4330.DBX79.1, 500 ms
   "2080SP241Y01.FP_CMD.Reset" : Bool AT %DB4330.DBX79.7, 500 ms
   "2080SP241Y01.FP_SHOW.PB_Auto" : Bool AT %DB4330.DBX88.0, 500 ms
   "2080SP241Y01.FP_SHOW.PB_Local" : Bool AT %DB4330.DBX88.1, 500 ms
   "2080SP241Y01.FP_SHOW.PB_Manual" : Bool AT %DB4330.DBX88.2, 500 ms
   "2080SP241Y01.FP_SHOW.PB_Start1" : Bool AT %DB4330.DBX88.3, 500 ms
   "2080SP241Y01.FP_SHOW.PB_Start2" : Bool AT %DB4330.DBX88.4, 500 ms
   "2080SP241Y01.FP_SHOW.PB_Start3" : Bool AT %DB4330.DBX88.5, 500 ms
   "2080SP241Y01.FP_SHOW.PB_Stop" : Bool AT %DB4330.DBX88.6, 500 ms
   "2080SP241Y01.FP_SHOW.PB_Test" : Bool AT %DB4330.DBX88.7, 500 ms
   "2080SP241Y01.FP_SHOW.PB_QStop" : Bool AT %DB4330.DBX89.0, 500 ms
   "2080SP241Y01.FP_SHOW.AI1" : Bool AT %DB4330.DBX89.1, 500 ms
   "2080SP241Y01.FP_SHOW.AI2" : Bool AT %DB4330.DBX89.2, 500 ms
   "2080SP241Y01.FP_SHOW.AI3" : Bool AT %DB4330.DBX89.3, 500 ms
   "2080SP241Y01.FP_SHOW.RDY" : Bool AT %DB4330.DBX89.4, 500 ms
   "2080SP241Y01.FP_SHOW.OVL" : Bool AT %DB4330.DBX89.5, 500 ms
   "2080SP241Y01.FP_SHOW.REM" : Bool AT %DB4330.DBX89.7, 500 ms
   "2080SP241Y01.FP_SHOW.SSW" : Bool AT %DB4330.DBX90.0, 500 ms
   "2080SP241Y01.FP_SHOW.DRDY" : Bool AT %DB4330.DBX90.1, 500 ms
   "2080SP241Y01.FP_SHOW.GFA" : Bool AT %DB4330.DBX90.2, 500 ms
   "2080SP241Y01.FP_SHOW.GWA" : Bool AT %DB4330.DBX90.3, 500 ms
   "2080SP241Y01.FP_SHOW.BUSF" : Bool AT %DB4330.DBX90.4, 500 ms
   "2080SP241Y01.FP_SHOW.UTEST" : Bool AT %DB4330.DBX90.6, 500 ms
   "2080SP241Y01.FP_SHOW.ACK" : Bool AT %DB4330.DBX90.7, 500 ms
   "2080SP241Y01.FP_SHOW.LSTR1" : Bool AT %DB4330.DBX91.0, 500 ms
   "2080SP241Y01.FP_SHOW.LSTR2" : Bool AT %DB4330.DBX91.1, 500 ms
   "2080SP241Y01.FP_SHOW.LSTR3" : Bool AT %DB4330.DBX91.2, 500 ms
   "2080SP241Y01.FP_SHOW.INTL3" : Bool AT %DB4330.DBX91.3, 500 ms
   "2080SP241Y01.FP_SHOW.CON3" : Bool AT %DB4330.DBX91.4, 500 ms
   "2080SP241Y01.FP_SHOW.PREQ3" : Bool AT %DB4330.DBX91.5, 500 ms
   "2080SP241Y01.FP_SHOW.LSP1" : Bool AT %DB4330.DBX91.6, 500 ms
   "2080SP241Y01.FP_SHOW.LSP2" : Bool AT %DB4330.DBX91.7, 500 ms
   "2080SP241Y01.FP_SHOW.LSP3" : Bool AT %DB4330.DBX92.0, 500 ms
   "2080SP241Y01.FP_SHOW.RunTime" : Bool AT %DB4330.DBX92.1, 500 ms
   "2080SP241Y01.FP_SHOW.LimitDrift" : Bool AT %DB4330.DBX92.2, 500 ms
   "2080SP241Y01.FP_SHOW.PB_Reset" : Bool AT %DB4330.DBX92.3, 500 ms
   "2080SP241Y01.FP_SHOW.POS3" : Bool AT %DB4330.DBX92.4, 500 ms
   "2080SP241Y01.FP_DIM.Auto" : Bool AT %DB4330.DBX86.0, 500 ms
   "2080SP241Y01.FP_DIM.Local" : Bool AT %DB4330.DBX86.1, 500 ms
   "2080SP241Y01.FP_DIM.Manual" : Bool AT %DB4330.DBX86.2, 500 ms
   "2080SP241Y01.FP_DIM.Start1" : Bool AT %DB4330.DBX86.3, 500 ms
   "2080SP241Y01.FP_DIM.Start2" : Bool AT %DB4330.DBX86.4, 500 ms
   "2080SP241Y01.FP_DIM.Start3" : Bool AT %DB4330.DBX86.5, 500 ms
   "2080SP241Y01.FP_DIM.Stop" : Bool AT %DB4330.DBX86.6, 500 ms
   "2080SP241Y01.FP_DIM.Test" : Bool AT %DB4330.DBX86.7, 500 ms
   "2080SP241Y01.FP_DIM.QStop" : Bool AT %DB4330.DBX87.0, 500 ms
   "2080SP241Y01.FP_DIM.Reset" : Bool AT %DB4330.DBX87.1, 500 ms
   "2080SP241Y01.FP_CMD.Start3" : Bool AT %DB4330.DBX79.5, 500 ms
   "2080SP241Y01.DI.SEL" : Bool AT %DB4330.DBX2.0, 500 ms
   "2080SP241Y01.DI.PREQ1" : Bool AT %DB4330.DBX2.1, 500 ms
   "2080SP241Y01.DI.PREQ2" : Bool AT %DB4330.DBX2.2, 500 ms
   "2080SP241Y01.DI.PREQ3" : Bool AT %DB4330.DBX2.3, 500 ms
   "2080SP241Y01.DI.RDY" : Bool AT %DB4330.DBX2.4, 500 ms
   "2080SP241Y01.DI.OVL" : Bool AT %DB4330.DBX2.5, 500 ms
   "2080SP241Y01.DI.LSP1" : Bool AT %DB4330.DBX2.6, 500 ms
   "2080SP241Y01.DI.LSP2" : Bool AT %DB4330.DBX2.7, 500 ms
   "2080SP241Y01.DI.LSP3" : Bool AT %DB4330.DBX3.0, 500 ms
   "2080SP241Y01.DI.LSTR1" : Bool AT %DB4330.DBX3.1, 500 ms
   "2080SP241Y01.DI.LSTR2" : Bool AT %DB4330.DBX3.2, 500 ms
   "2080SP241Y01.DI.LSTR3" : Bool AT %DB4330.DBX3.3, 500 ms
   "2080SP241Y01.DI.REM" : Bool AT %DB4330.DBX3.4, 500 ms
   "2080SP241Y01.DI.SSW" : Bool AT %DB4330.DBX3.5, 500 ms
   "2080SP241Y01.DI.DRDY" : Bool AT %DB4330.DBX3.6, 500 ms
   "2080SP241Y01.DI.GFA" : Bool AT %DB4330.DBX3.7, 500 ms
   "2080SP241Y01.DI.GWA" : Bool AT %DB4330.DBX4.0, 500 ms
   "2080SP241Y01.DI.BUSF" : Bool AT %DB4330.DBX4.1, 500 ms
   "2080SP241Y01.DI.UTEST" : Bool AT %DB4330.DBX4.2, 500 ms
   "2080SP241Y01.DI.ACK" : Bool AT %DB4330.DBX4.3, 500 ms
   "2080SP241Y01.DQ.CON1" : Bool AT %DB4330.DBX28.0, 500 ms
   "2080SP241Y01.DQ.CON2" : Bool AT %DB4330.DBX28.1, 500 ms
   "2080SP241Y01.DQ.CON3" : Bool AT %DB4330.DBX28.2, 500 ms
   "2080SP241Y01.DQ.LAMP1" : Bool AT %DB4330.DBX28.3, 500 ms
   "2080SP241Y01.DQ.LAMP2" : Bool AT %DB4330.DBX28.4, 500 ms
   "2080SP241Y01.DQ.LAMP3" : Bool AT %DB4330.DBX28.5, 500 ms
   "2080SP241Y01.DQ.SACK" : Bool AT %DB4330.DBX28.6, 500 ms
   "2080SP241Y01.DQ.POS1" : Bool AT %DB4330.DBX28.7, 500 ms
   "2080SP241Y01.DQ.POS2" : Bool AT %DB4330.DBX29.0, 500 ms
   "2080SP241Y01.DQ.POS3" : Bool AT %DB4330.DBX29.1, 500 ms
   "2080SP241Y01.DQ.OK" : Bool AT %DB4330.DBX29.2, 500 ms
   "2080SP241Y01.DQ.LOC" : Bool AT %DB4330.DBX29.3, 500 ms
   "2080SP241Y01.DQ.MAN" : Bool AT %DB4330.DBX29.4, 500 ms
   "2080SP241Y01.DQ.AUT" : Bool AT %DB4330.DBX29.5, 500 ms
   "2080SP241Y01.DQ.SS" : Bool AT %DB4330.DBX29.6, 500 ms
   "2080SP241Y01.DQ.RES" : Bool AT %DB4330.DBX29.7, 500 ms
   "2080SP241Y01.DQ.TESTP" : Bool AT %DB4330.DBX30.0, 500 ms
   "2080SP241Y01.DQ.ASTW" : Bool AT %DB4330.DBX30.1, 500 ms
   "2080SP241Y01.DQ.AL_SUPR" : Bool AT %DB4330.DBX30.2, 500 ms
   "2080SP241Y01.FP_PARM.StartWarn_Pre" : Int AT %DB4330.DBW94, 500 ms
   "2080SP241Y01.FP_PARM.StartWarn_Acc" : Int AT %DB4330.DBW96, 500 ms
   "2080SP241Y01.FP_PARM.RunTime_Pre" : Int AT %DB4330.DBW98, 500 ms
   "2080SP241Y01.FP_PARM.RunTime_Acc" : Int AT %DB4330.DBW100, 500 ms
   "2080SP241Y01.FP_PARM.DriftingTime_Pre" : Int AT %DB4330.DBW102, 500 ms
   "2080SP241Y01.FP_PARM.DriftingTime_Acc" : Int AT %DB4330.DBW104, 500 ms
   "2080SP241Y01.FP_PARM.DelayStart_Pre" : Int AT %DB4330.DBW106, 500 ms
   "2080SP241Y01.FP_PARM.DelayStart_Acc" : Int AT %DB4330.DBW108, 500 ms
   "2080SP241Y01.FP_PARM.DelayStop_Pre" : Int AT %DB4330.DBW110, 500 ms
   "2080SP241Y01.FP_PARM.DelayStop_Acc" : Int AT %DB4330.DBW112, 500 ms
   "2080SP241Y01.FP_PARM.AI1_Max" : Real AT %DB4330.DBD114, 500 ms
   "2080SP241Y01.FP_PARM.AI1_Min" : Real AT %DB4330.DBD118, 500 ms
   "2080SP241Y01.FP_PARM.AI2_Max" : Real AT %DB4330.DBD122, 500 ms
   "2080SP241Y01.FP_PARM.AI2_Min" : Real AT %DB4330.DBD126, 500 ms
   "2080SP241Y01.FP_PARM.AI3_Max" : Real AT %DB4330.DBD130, 500 ms
   "2080SP241Y01.FP_PARM.AI3_Min" : Real AT %DB4330.DBD134, 500 ms
   "2080SP241Y01.FP_PARM.AO1a_Max" : Real AT %DB4330.DBD138, 500 ms
   "2080SP241Y01.FP_PARM.AO1a_Min" : Real AT %DB4330.DBD142, 500 ms
   "2080SP241Y01.FP_PARM.AO2a_Max" : Real AT %DB4330.DBD146, 500 ms
   "2080SP241Y01.FP_PARM.AO2a_Min" : Real AT %DB4330.DBD150, 500 ms
   "2080SP241Y01.FP_PARM.AO3a_Max" : Real AT %DB4330.DBD154, 500 ms
   "2080SP241Y01.FP_PARM.AO3a_Min" : Real AT %DB4330.DBD158, 500 ms
   "2080SP241Y01.FP_PARM.AO1b_Max" : Real AT %DB4330.DBD162, 500 ms
   "2080SP241Y01.FP_PARM.AO1b_Min" : Real AT %DB4330.DBD166, 500 ms
   "2080SP241Y01.FP_PARM.AO2b_Max" : Real AT %DB4330.DBD170, 500 ms
   "2080SP241Y01.FP_PARM.AO2b_Min" : Real AT %DB4330.DBD174, 500 ms
   "2080SP241Y01.FP_PARM.AO3b_Max" : Real AT %DB4330.DBD178, 500 ms
   "2080SP241Y01.FP_PARM.AO3b_Min" : Real AT %DB4330.DBD182, 500 ms
   "2080SP241Y01.FP_SEL.STW_AutoStart" : Bool AT %DB4330.DBX80.0, 500 ms
   "2080SP241Y01.FP_SEL.STW_Local" : Bool AT %DB4330.DBX80.1, 500 ms
   "2080SP241Y01.FP_SEL.STW_Manual" : Bool AT %DB4330.DBX80.2, 500 ms
   "2080SP241Y01.FP_SEL.STW_Single" : Bool AT %DB4330.DBX80.3, 500 ms
   "2080SP241Y01.FP_SEL.Type_2Pos" : Bool AT %DB4330.DBX80.4, 500 ms
   "2080SP241Y01.FP_SEL.Type_3Pos" : Bool AT %DB4330.DBX80.5, 500 ms
   "2080SP241Y01.FP_SEL.Type_Indication" : Bool AT %DB4330.DBX80.6, 500 ms
   "2080SP241Y01.FP_SEL.Type_NoLimit" : Bool AT %DB4330.DBX80.7, 500 ms
   "2080SP241Y01.FP_SEL.Type_ConstantCmd" : Bool AT %DB4330.DBX81.0, 500 ms
   "2080SP241Y01.FP_SEL.Type_PulseCmd" : Bool AT %DB4330.DBX81.1, 500 ms
   "2080SP241Y01.FP_SEL.ParentSupress" : Bool AT %DB4330.DBX81.2, 500 ms
   "2080SP241Y01.FP_SEL.ParentCollection" : Bool AT %DB4330.DBX81.3, 500 ms
   "2080SP241Y01.FP_SEL.INCH_Man" : Bool AT %DB4330.DBX81.4, 500 ms
   "2080SP241Y01.FP_SEL.INCH_Loc" : Bool AT %DB4330.DBX81.5, 500 ms
   "2080SP241Y01.FP_SEL.OutOfSevice" : Bool AT %DB4330.DBX81.6, 500 ms
   "2080SP241Y01.FP_SEL.WarningDrive" : Bool AT %DB4330.DBX81.7, 500 ms
   "2080SP241Y01.FP_SEL.Park_CurrPos" : Bool AT %DB4330.DBX82.0, 500 ms
   "2080SP241Y01.FP_SEL.Park_Pos1" : Bool AT %DB4330.DBX82.1, 500 ms
   "2080SP241Y01.FP_SEL.Park_Pos2" : Bool AT %DB4330.DBX82.2, 500 ms
   "2080SP241Y01.FP_SEL.Park_Pos3" : Bool AT %DB4330.DBX82.3, 500 ms
   "2080SP241Y01.FP_SEL.GroupMode" : Bool AT %DB4330.DBX82.4, 500 ms
   "2080SP241Y01.FP_SEL.GroupCtrl" : Bool AT %DB4330.DBX82.5, 500 ms
   "2080SP241Y01.FP_EN.Mode_Auto" : Bool AT %DB4330.DBX84.0, 500 ms
   "2080SP241Y01.FP_EN.Mode_Man" : Bool AT %DB4330.DBX84.1, 500 ms
   "2080SP241Y01.FP_EN.Mode_Loc" : Bool AT %DB4330.DBX84.2, 500 ms
   "2080SP241Y01.FP_EN.Mode_Test" : Bool AT %DB4330.DBX84.3, 500 ms
   "2080SP241Y01.FP_EN.Mode_SS_Field" : Bool AT %DB4330.DBX84.4, 500 ms
   "2080SP241Y01.FP_EN.Mode_SS_FP" : Bool AT %DB4330.DBX84.5, 500 ms
   "2080SP241Y01.FP_EN.PB_QStop" : Bool AT %DB4330.DBX84.6, 500 ms
   "2080SP241Y01.BlockInfo" : Array [0..4] of Int AT %DB4330.DBX68.0, 500 ms
   "2080SP241Y01.ParentInfo" : TextRef, internal   // Имя родителя для попап окна, вкладка инфо. При експорте из ECS через скрипт заполняется автоматически, если теги копируются в ручную то требуется в ручную задатать свойство Start Value
   "2080SP241Y01.MSW" : DWord AT %DB4330.DBD56, 500 ms

HMI tags "2080SP242Y01"
   "2080SP242Y01.DefaultText" : TextRef, internal   // Заголовок POPUP окна. При експорте из ECS через скрипт заполняется автоматически, если теги копируются в ручную то требуется в ручную задатать свойство Start Value
   "2080SP242Y01.StatusWork" : Int AT %DB4329.DBW458, 500 ms
   "2080SP242Y01.ModePointer" : Int AT %DB4329.DBW460, 500 ms
   "2080SP242Y01.FP_CMD.Start1" : Bool AT %DB4329.DBX79.3, 500 ms
   "2080SP242Y01.FP_CMD.Start2" : Bool AT %DB4329.DBX79.4, 500 ms
   "2080SP242Y01.FP_CMD.Stop" : Bool AT %DB4329.DBX79.6, 500 ms
   "2080SP242Y01.FP_CMD.AckAlarm" : Bool AT %DB4329.DBX78.7, 500 ms
   "2080SP242Y01.FP_CMD.Auto" : Bool AT %DB4329.DBX79.0, 500 ms
   "2080SP242Y01.FP_CMD.Local" : Bool AT %DB4329.DBX79.2, 500 ms
   "2080SP242Y01.FP_CMD.Manual" : Bool AT %DB4329.DBX79.1, 500 ms
   "2080SP242Y01.FP_CMD.Reset" : Bool AT %DB4329.DBX79.7, 500 ms
   "2080SP242Y01.FP_SHOW.PB_Auto" : Bool AT %DB4329.DBX88.0, 500 ms
   "2080SP242Y01.FP_SHOW.PB_Local" : Bool AT %DB4329.DBX88.1, 500 ms
   "2080SP242Y01.FP_SHOW.PB_Manual" : Bool AT %DB4329.DBX88.2, 500 ms
   "2080SP242Y01.FP_SHOW.PB_Start1" : Bool AT %DB4329.DBX88.3, 500 ms
   "2080SP242Y01.FP_SHOW.PB_Start2" : Bool AT %DB4329.DBX88.4, 500 ms
   "2080SP242Y01.FP_SHOW.PB_Start3" : Bool AT %DB4329.DBX88.5, 500 ms
   "2080SP242Y01.FP_SHOW.PB_Stop" : Bool AT %DB4329.DBX88.6, 500 ms
   "2080SP242Y01.FP_SHOW.PB_Test" : Bool AT %DB4329.DBX88.7, 500 ms
   "2080SP242Y01.FP_SHOW.PB_QStop" : Bool AT %DB4329.DBX89.0, 500 ms
   "2080SP242Y01.FP_SHOW.AI1" : Bool AT %DB4329.DBX89.1, 500 ms
   "2080SP242Y01.FP_SHOW.AI2" : Bool AT %DB4329.DBX89.2, 500 ms
   "2080SP242Y01.FP_SHOW.AI3" : Bool AT %DB4329.DBX89.3, 500 ms
   "2080SP242Y01.FP_SHOW.RDY" : Bool AT %DB4329.DBX89.4, 500 ms
   "2080SP242Y01.FP_SHOW.OVL" : Bool AT %DB4329.DBX89.5, 500 ms
   "2080SP242Y01.FP_SHOW.REM" : Bool AT %DB4329.DBX89.7, 500 ms
   "2080SP242Y01.FP_SHOW.SSW" : Bool AT %DB4329.DBX90.0, 500 ms
   "2080SP242Y01.FP_SHOW.DRDY" : Bool AT %DB4329.DBX90.1, 500 ms
   "2080SP242Y01.FP_SHOW.GFA" : Bool AT %DB4329.DBX90.2, 500 ms
   "2080SP242Y01.FP_SHOW.GWA" : Bool AT %DB4329.DBX90.3, 500 ms
   "2080SP242Y01.FP_SHOW.BUSF" : Bool AT %DB4329.DBX90.4, 500 ms
   "2080SP242Y01.FP_SHOW.UTEST" : Bool AT %DB4329.DBX90.6, 500 ms
   "2080SP242Y01.FP_SHOW.ACK" : Bool AT %DB4329.DBX90.7, 500 ms
   "2080SP242Y01.FP_SHOW.LSTR1" : Bool AT %DB4329.DBX91.0, 500 ms
   "2080SP242Y01.FP_SHOW.LSTR2" : Bool AT %DB4329.DBX91.1, 500 ms
   "2080SP242Y01.FP_SHOW.LSTR3" : Bool AT %DB4329.DBX91.2, 500 ms
   "2080SP242Y01.FP_SHOW.INTL3" : Bool AT %DB4329.DBX91.3, 500 ms
   "2080SP242Y01.FP_SHOW.CON3" : Bool AT %DB4329.DBX91.4, 500 ms
   "2080SP242Y01.FP_SHOW.PREQ3" : Bool AT %DB4329.DBX91.5, 500 ms
   "2080SP242Y01.FP_SHOW.LSP1" : Bool AT %DB4329.DBX91.6, 500 ms
   "2080SP242Y01.FP_SHOW.LSP2" : Bool AT %DB4329.DBX91.7, 500 ms
   "2080SP242Y01.FP_SHOW.LSP3" : Bool AT %DB4329.DBX92.0, 500 ms
   "2080SP242Y01.FP_SHOW.RunTime" : Bool AT %DB4329.DBX92.1, 500 ms
   "2080SP242Y01.FP_SHOW.LimitDrift" : Bool AT %DB4329.DBX92.2, 500 ms
   "2080SP242Y01.FP_SHOW.PB_Reset" : Bool AT %DB4329.DBX92.3, 500 ms
   "2080SP242Y01.FP_SHOW.POS3" : Bool AT %DB4329.DBX92.4, 500 ms
   "2080SP242Y01.FP_DIM.Auto" : Bool AT %DB4329.DBX86.0, 500 ms
   "2080SP242Y01.FP_DIM.Local" : Bool AT %DB4329.DBX86.1, 500 ms
   "2080SP242Y01.FP_DIM.Manual" : Bool AT %DB4329.DBX86.2, 500 ms
   "2080SP242Y01.FP_DIM.Start1" : Bool AT %DB4329.DBX86.3, 500 ms
   "2080SP242Y01.FP_DIM.Start2" : Bool AT %DB4329.DBX86.4, 500 ms
   "2080SP242Y01.FP_DIM.Start3" : Bool AT %DB4329.DBX86.5, 500 ms
   "2080SP242Y01.FP_DIM.Stop" : Bool AT %DB4329.DBX86.6, 500 ms
   "2080SP242Y01.FP_DIM.Test" : Bool AT %DB4329.DBX86.7, 500 ms
   "2080SP242Y01.FP_DIM.QStop" : Bool AT %DB4329.DBX87.0, 500 ms
   "2080SP242Y01.FP_DIM.Reset" : Bool AT %DB4329.DBX87.1, 500 ms
   "2080SP242Y01.FP_CMD.Start3" : Bool AT %DB4329.DBX79.5, 500 ms
   "2080SP242Y01.DI.SEL" : Bool AT %DB4329.DBX2.0, 500 ms
   "2080SP242Y01.DI.PREQ1" : Bool AT %DB4329.DBX2.1, 500 ms
   "2080SP242Y01.DI.PREQ2" : Bool AT %DB4329.DBX2.2, 500 ms
   "2080SP242Y01.DI.PREQ3" : Bool AT %DB4329.DBX2.3, 500 ms
   "2080SP242Y01.DI.RDY" : Bool AT %DB4329.DBX2.4, 500 ms
   "2080SP242Y01.DI.OVL" : Bool AT %DB4329.DBX2.5, 500 ms
   "2080SP242Y01.DI.LSP1" : Bool AT %DB4329.DBX2.6, 500 ms
   "2080SP242Y01.DI.LSP2" : Bool AT %DB4329.DBX2.7, 500 ms
   "2080SP242Y01.DI.LSP3" : Bool AT %DB4329.DBX3.0, 500 ms
   "2080SP242Y01.DI.LSTR1" : Bool AT %DB4329.DBX3.1, 500 ms
   "2080SP242Y01.DI.LSTR2" : Bool AT %DB4329.DBX3.2, 500 ms
   "2080SP242Y01.DI.LSTR3" : Bool AT %DB4329.DBX3.3, 500 ms
   "2080SP242Y01.DI.REM" : Bool AT %DB4329.DBX3.4, 500 ms
   "2080SP242Y01.DI.SSW" : Bool AT %DB4329.DBX3.5, 500 ms
   "2080SP242Y01.DI.DRDY" : Bool AT %DB4329.DBX3.6, 500 ms
   "2080SP242Y01.DI.GFA" : Bool AT %DB4329.DBX3.7, 500 ms
   "2080SP242Y01.DI.GWA" : Bool AT %DB4329.DBX4.0, 500 ms
   "2080SP242Y01.DI.BUSF" : Bool AT %DB4329.DBX4.1, 500 ms
   "2080SP242Y01.DI.UTEST" : Bool AT %DB4329.DBX4.2, 500 ms
   "2080SP242Y01.DI.ACK" : Bool AT %DB4329.DBX4.3, 500 ms
   "2080SP242Y01.DQ.CON1" : Bool AT %DB4329.DBX28.0, 500 ms
   "2080SP242Y01.DQ.CON2" : Bool AT %DB4329.DBX28.1, 500 ms
   "2080SP242Y01.DQ.CON3" : Bool AT %DB4329.DBX28.2, 500 ms
   "2080SP242Y01.DQ.LAMP1" : Bool AT %DB4329.DBX28.3, 500 ms
   "2080SP242Y01.DQ.LAMP2" : Bool AT %DB4329.DBX28.4, 500 ms
   "2080SP242Y01.DQ.LAMP3" : Bool AT %DB4329.DBX28.5, 500 ms
   "2080SP242Y01.DQ.SACK" : Bool AT %DB4329.DBX28.6, 500 ms
   "2080SP242Y01.DQ.POS1" : Bool AT %DB4329.DBX28.7, 500 ms
   "2080SP242Y01.DQ.POS2" : Bool AT %DB4329.DBX29.0, 500 ms
   "2080SP242Y01.DQ.POS3" : Bool AT %DB4329.DBX29.1, 500 ms
   "2080SP242Y01.DQ.OK" : Bool AT %DB4329.DBX29.2, 500 ms
   "2080SP242Y01.DQ.LOC" : Bool AT %DB4329.DBX29.3, 500 ms
   "2080SP242Y01.DQ.MAN" : Bool AT %DB4329.DBX29.4, 500 ms
   "2080SP242Y01.DQ.AUT" : Bool AT %DB4329.DBX29.5, 500 ms
   "2080SP242Y01.DQ.SS" : Bool AT %DB4329.DBX29.6, 500 ms
   "2080SP242Y01.DQ.RES" : Bool AT %DB4329.DBX29.7, 500 ms
   "2080SP242Y01.DQ.TESTP" : Bool AT %DB4329.DBX30.0, 500 ms
   "2080SP242Y01.DQ.ASTW" : Bool AT %DB4329.DBX30.1, 500 ms
   "2080SP242Y01.DQ.AL_SUPR" : Bool AT %DB4329.DBX30.2, 500 ms
   "2080SP242Y01.FP_PARM.StartWarn_Pre" : Int AT %DB4329.DBW94, 500 ms
   "2080SP242Y01.FP_PARM.StartWarn_Acc" : Int AT %DB4329.DBW96, 500 ms
   "2080SP242Y01.FP_PARM.RunTime_Pre" : Int AT %DB4329.DBW98, 500 ms
   "2080SP242Y01.FP_PARM.RunTime_Acc" : Int AT %DB4329.DBW100, 500 ms
   "2080SP242Y01.FP_PARM.DriftingTime_Pre" : Int AT %DB4329.DBW102, 500 ms
   "2080SP242Y01.FP_PARM.DriftingTime_Acc" : Int AT %DB4329.DBW104, 500 ms
   "2080SP242Y01.FP_PARM.DelayStart_Pre" : Int AT %DB4329.DBW106, 500 ms
   "2080SP242Y01.FP_PARM.DelayStart_Acc" : Int AT %DB4329.DBW108, 500 ms
   "2080SP242Y01.FP_PARM.DelayStop_Pre" : Int AT %DB4329.DBW110, 500 ms
   "2080SP242Y01.FP_PARM.DelayStop_Acc" : Int AT %DB4329.DBW112, 500 ms
   "2080SP242Y01.FP_PARM.AI1_Max" : Real AT %DB4329.DBD114, 500 ms
   "2080SP242Y01.FP_PARM.AI1_Min" : Real AT %DB4329.DBD118, 500 ms
   "2080SP242Y01.FP_PARM.AI2_Max" : Real AT %DB4329.DBD122, 500 ms
   "2080SP242Y01.FP_PARM.AI2_Min" : Real AT %DB4329.DBD126, 500 ms
   "2080SP242Y01.FP_PARM.AI3_Max" : Real AT %DB4329.DBD130, 500 ms
   "2080SP242Y01.FP_PARM.AI3_Min" : Real AT %DB4329.DBD134, 500 ms
   "2080SP242Y01.FP_PARM.AO1a_Max" : Real AT %DB4329.DBD138, 500 ms
   "2080SP242Y01.FP_PARM.AO1a_Min" : Real AT %DB4329.DBD142, 500 ms
   "2080SP242Y01.FP_PARM.AO2a_Max" : Real AT %DB4329.DBD146, 500 ms
   "2080SP242Y01.FP_PARM.AO2a_Min" : Real AT %DB4329.DBD150, 500 ms
   "2080SP242Y01.FP_PARM.AO3a_Max" : Real AT %DB4329.DBD154, 500 ms
   "2080SP242Y01.FP_PARM.AO3a_Min" : Real AT %DB4329.DBD158, 500 ms
   "2080SP242Y01.FP_PARM.AO1b_Max" : Real AT %DB4329.DBD162, 500 ms
   "2080SP242Y01.FP_PARM.AO1b_Min" : Real AT %DB4329.DBD166, 500 ms
   "2080SP242Y01.FP_PARM.AO2b_Max" : Real AT %DB4329.DBD170, 500 ms
   "2080SP242Y01.FP_PARM.AO2b_Min" : Real AT %DB4329.DBD174, 500 ms
   "2080SP242Y01.FP_PARM.AO3b_Max" : Real AT %DB4329.DBD178, 500 ms
   "2080SP242Y01.FP_PARM.AO3b_Min" : Real AT %DB4329.DBD182, 500 ms
   "2080SP242Y01.FP_SEL.STW_AutoStart" : Bool AT %DB4329.DBX80.0, 500 ms
   "2080SP242Y01.FP_SEL.STW_Local" : Bool AT %DB4329.DBX80.1, 500 ms
   "2080SP242Y01.FP_SEL.STW_Manual" : Bool AT %DB4329.DBX80.2, 500 ms
   "2080SP242Y01.FP_SEL.STW_Single" : Bool AT %DB4329.DBX80.3, 500 ms
   "2080SP242Y01.FP_SEL.Type_2Pos" : Bool AT %DB4329.DBX80.4, 500 ms
   "2080SP242Y01.FP_SEL.Type_3Pos" : Bool AT %DB4329.DBX80.5, 500 ms
   "2080SP242Y01.FP_SEL.Type_Indication" : Bool AT %DB4329.DBX80.6, 500 ms
   "2080SP242Y01.FP_SEL.Type_NoLimit" : Bool AT %DB4329.DBX80.7, 500 ms
   "2080SP242Y01.FP_SEL.Type_ConstantCmd" : Bool AT %DB4329.DBX81.0, 500 ms
   "2080SP242Y01.FP_SEL.Type_PulseCmd" : Bool AT %DB4329.DBX81.1, 500 ms
   "2080SP242Y01.FP_SEL.ParentSupress" : Bool AT %DB4329.DBX81.2, 500 ms
   "2080SP242Y01.FP_SEL.ParentCollection" : Bool AT %DB4329.DBX81.3, 500 ms
   "2080SP242Y01.FP_SEL.INCH_Man" : Bool AT %DB4329.DBX81.4, 500 ms
   "2080SP242Y01.FP_SEL.INCH_Loc" : Bool AT %DB4329.DBX81.5, 500 ms
   "2080SP242Y01.FP_SEL.OutOfSevice" : Bool AT %DB4329.DBX81.6, 500 ms
   "2080SP242Y01.FP_SEL.WarningDrive" : Bool AT %DB4329.DBX81.7, 500 ms
   "2080SP242Y01.FP_SEL.Park_CurrPos" : Bool AT %DB4329.DBX82.0, 500 ms
   "2080SP242Y01.FP_SEL.Park_Pos1" : Bool AT %DB4329.DBX82.1, 500 ms
   "2080SP242Y01.FP_SEL.Park_Pos2" : Bool AT %DB4329.DBX82.2, 500 ms
   "2080SP242Y01.FP_SEL.Park_Pos3" : Bool AT %DB4329.DBX82.3, 500 ms
   "2080SP242Y01.FP_SEL.GroupMode" : Bool AT %DB4329.DBX82.4, 500 ms
   "2080SP242Y01.FP_SEL.GroupCtrl" : Bool AT %DB4329.DBX82.5, 500 ms
   "2080SP242Y01.FP_EN.Mode_Auto" : Bool AT %DB4329.DBX84.0, 500 ms
   "2080SP242Y01.FP_EN.Mode_Man" : Bool AT %DB4329.DBX84.1, 500 ms
   "2080SP242Y01.FP_EN.Mode_Loc" : Bool AT %DB4329.DBX84.2, 500 ms
   "2080SP242Y01.FP_EN.Mode_Test" : Bool AT %DB4329.DBX84.3, 500 ms
   "2080SP242Y01.FP_EN.Mode_SS_Field" : Bool AT %DB4329.DBX84.4, 500 ms
   "2080SP242Y01.FP_EN.Mode_SS_FP" : Bool AT %DB4329.DBX84.5, 500 ms
   "2080SP242Y01.FP_EN.PB_QStop" : Bool AT %DB4329.DBX84.6, 500 ms
   "2080SP242Y01.BlockInfo" : Array [0..4] of Int AT %DB4329.DBX68.0, 500 ms
   "2080SP242Y01.ParentInfo" : TextRef, internal   // Имя родителя для попап окна, вкладка инфо. При експорте из ECS через скрипт заполняется автоматически, если теги копируются в ручную то требуется в ручную задатать свойство Start Value
   "2080SP242Y01.MSW" : DWord AT %DB4329.DBD56, 500 ms

HMI tags "2080SP241U01"
   "2080SP241U01.AI1" : Real AT %DB4303.DBD6, 500 ms
   "2080SP241U01.AI2" : Real AT %DB4303.DBD10, 500 ms
   "2080SP241U01.AI3" : Real AT %DB4303.DBD14, 500 ms
   "2080SP241U01.AO1a" : Real AT %DB4303.DBD34, 500 ms
   "2080SP241U01.AO1b" : Real AT %DB4303.DBD38, 500 ms
   "2080SP241U01.AO2a" : Real AT %DB4303.DBD42, 500 ms
   "2080SP241U01.AO2b" : Real AT %DB4303.DBD42, 500 ms
   "2080SP241U01.AO3a" : Real AT %DB4303.DBD50, 500 ms
   "2080SP241U01.AO3b" : Real AT %DB4303.DBD46, 500 ms
   "2080SP241U01.BlockInfo" : Array [0..4] of Int AT %DB4303.DBX74.0, 500 ms
   "2080SP241U01.DefaultText" : TextRef, internal   // Заголовок POPUP окна. При експорте из ECS через скрипт заполняется автоматически, если теги копируются в ручную то требуется в ручную задатать свойство Start Value
   "2080SP241U01.DI.ACK" : Bool AT %DB4303.DBX5.3, 500 ms
   "2080SP241U01.DI.ASTR" : Bool AT %DB4303.DBX2.1, 500 ms
   "2080SP241U01.DI.BUSF" : Bool AT %DB4303.DBX4.5, 500 ms
   "2080SP241U01.DI.DIR" : Bool AT %DB4303.DBX2.2, 500 ms
   "2080SP241U01.DI.DOPR" : Bool AT %DB4303.DBX4.6, 500 ms
   "2080SP241U01.DI.DRDY" : Bool AT %DB4303.DBX3.6, 500 ms
   "2080SP241U01.DI.DTEST" : Bool AT %DB4303.DBX4.7, 500 ms
   "2080SP241U01.DI.EARTH" : Bool AT %DB4303.DBX4.1, 500 ms
   "2080SP241U01.DI.ES" : Bool AT %DB4303.DBX5.2, 500 ms
   "2080SP241U01.DI.GFA" : Bool AT %DB4303.DBX4.3, 500 ms
   "2080SP241U01.DI.GWA" : Bool AT %DB4303.DBX4.4, 500 ms
   "2080SP241U01.DI.LSTP" : Bool AT %DB4303.DBX3.2, 500 ms
   "2080SP241U01.DI.LSTR1" : Bool AT %DB4303.DBX3.0, 500 ms
   "2080SP241U01.DI.LSTR2" : Bool AT %DB4303.DBX3.1, 500 ms
   "2080SP241U01.DI.MCC" : Bool AT %DB4303.DBX2.3, 500 ms
   "2080SP241U01.DI.MD" : Bool AT %DB4303.DBX3.7, 500 ms
   "2080SP241U01.DI.OVL" : Bool AT %DB4303.DBX2.5, 500 ms
   "2080SP241U01.DI.RDY" : Bool AT %DB4303.DBX2.4, 500 ms
   "2080SP241U01.DI.REM" : Bool AT %DB4303.DBX3.3, 500 ms
   "2080SP241U01.DI.RET1" : Bool AT %DB4303.DBX2.6, 500 ms
   "2080SP241U01.DI.RET2" : Bool AT %DB4303.DBX2.7, 500 ms
   "2080SP241U01.DI.SEL" : Bool AT %DB4303.DBX2.0, 500 ms
   "2080SP241U01.DI.SFS" : Bool AT %DB4303.DBX5.0, 500 ms
   "2080SP241U01.DI.SLS" : Bool AT %DB4303.DBX5.1, 500 ms
   "2080SP241U01.DI.SSW" : Bool AT %DB4303.DBX3.4, 500 ms
   "2080SP241U01.DI.STALL" : Bool AT %DB4303.DBX4.0, 500 ms
   "2080SP241U01.DI.TFA" : Bool AT %DB4303.DBX3.5, 500 ms
   "2080SP241U01.DI.UBAL" : Bool AT %DB4303.DBX4.2, 500 ms
   "2080SP241U01.DQ.ASTW" : Bool AT %DB4303.DBX32.0, 500 ms
   "2080SP241U01.DQ.AUT" : Bool AT %DB4303.DBX31.4, 500 ms
   "2080SP241U01.DQ.CON1" : Bool AT %DB4303.DBX30.0, 500 ms
   "2080SP241U01.DQ.CON2" : Bool AT %DB4303.DBX30.1, 500 ms
   "2080SP241U01.DQ.LAMP1" : Bool AT %DB4303.DBX30.2, 500 ms
   "2080SP241U01.DQ.LAMP2" : Bool AT %DB4303.DBX30.3, 500 ms
   "2080SP241U01.DQ.LOC" : Bool AT %DB4303.DBX31.2, 500 ms
   "2080SP241U01.DQ.MAN" : Bool AT %DB4303.DBX31.3, 500 ms
   "2080SP241U01.DQ.OK" : Bool AT %DB4303.DBX31.1, 500 ms
   "2080SP241U01.DQ.RD1" : Bool AT %DB4303.DBX30.5, 500 ms
   "2080SP241U01.DQ.RD2" : Bool AT %DB4303.DBX30.6, 500 ms
   "2080SP241U01.DQ.RES" : Bool AT %DB4303.DBX31.6, 500 ms
   "2080SP241U01.DQ.RUN1" : Bool AT %DB4303.DBX30.7, 500 ms
   "2080SP241U01.DQ.RUN2" : Bool AT %DB4303.DBX31.0, 500 ms
   "2080SP241U01.DQ.SACK" : Bool AT %DB4303.DBX30.4, 500 ms
   "2080SP241U01.DQ.SS" : Bool AT %DB4303.DBX31.5, 500 ms
   "2080SP241U01.DQ.TESTP" : Bool AT %DB4303.DBX31.7, 500 ms
   "2080SP241U01.FP_CMD" : Int AT %DB4303.DBW84, 500 ms
   "2080SP241U01.FP_CMD.AckAlarm" : Bool AT %DB4303.DBX84.7, 500 ms
   "2080SP241U01.FP_CMD.Auto" : Bool AT %DB4303.DBX85.0, 500 ms
   "2080SP241U01.FP_CMD.Local" : Bool AT %DB4303.DBX85.2, 500 ms
   "2080SP241U01.FP_CMD.Manual" : Bool AT %DB4303.DBX85.1, 500 ms
   "2080SP241U01.FP_CMD.QuickStop" : Bool AT %DB4303.DBX84.0, 500 ms
   "2080SP241U01.FP_CMD.Reset" : Bool AT %DB4303.DBX85.6, 500 ms
   "2080SP241U01.FP_CMD.Start1" : Bool AT %DB4303.DBX85.3, 500 ms
   "2080SP241U01.FP_CMD.Start2" : Bool AT %DB4303.DBX85.4, 500 ms
   "2080SP241U01.FP_CMD.Stop" : Bool AT %DB4303.DBX85.5, 500 ms
   "2080SP241U01.FP_CMD.Test" : Bool AT %DB4303.DBX85.7, 500 ms
   "2080SP241U01.FP_DIM.Auto" : Bool AT %DB4303.DBX92.0, 500 ms
   "2080SP241U01.FP_DIM.FP_DIM" : Bool AT %DB4303.DBX92.0, 500 ms
   "2080SP241U01.FP_DIM.Local" : Bool AT %DB4303.DBX92.1, 500 ms
   "2080SP241U01.FP_DIM.Manual" : Bool AT %DB4303.DBX92.2, 500 ms
   "2080SP241U01.FP_DIM.QStop" : Bool AT %DB4303.DBX92.7, 500 ms
   "2080SP241U01.FP_DIM.Reset" : Bool AT %DB4303.DBX93.0, 500 ms
   "2080SP241U01.FP_DIM.Start1" : Bool AT %DB4303.DBX92.3, 500 ms
   "2080SP241U01.FP_DIM.Start2" : Bool AT %DB4303.DBX92.4, 500 ms
   "2080SP241U01.FP_DIM.Stop" : Bool AT %DB4303.DBX92.5, 500 ms
   "2080SP241U01.FP_DIM.TEst" : Bool AT %DB4303.DBX92.6, 500 ms
   "2080SP241U01.FP_DIM1" : Array [0..15] of Bool AT %DB4303.DBX92.0, 500 ms
   "2080SP241U01.FP_EN.Mode_Auto" : Bool AT %DB4303.DBX90.0, 500 ms
   "2080SP241U01.FP_EN.Mode_Loc" : Bool AT %DB4303.DBX90.2, 500 ms
   "2080SP241U01.FP_EN.Mode_Loc_1" : Bool AT %DB4303.DBX90.3, 500 ms
   "2080SP241U01.FP_EN.Mode_Man" : Bool AT %DB4303.DBX90.1, 500 ms
   "2080SP241U01.FP_EN.Mode_SS_Field" : Bool AT %DB4303.DBX90.4, 500 ms
   "2080SP241U01.FP_EN.Mode_SS_FP" : Bool AT %DB4303.DBX90.5, 500 ms
   "2080SP241U01.FP_EN.Mode_Test" : Bool AT %DB4303.DBX90.3, 500 ms
   "2080SP241U01.FP_EN.PB_QStop" : Bool AT %DB4303.DBX90.6, 500 ms
   "2080SP241U01.FP_PARM.AI1_Max" : Real AT %DB4303.DBD158, 500 ms
   "2080SP241U01.FP_PARM.AI1_Min" : Real AT %DB4303.DBD162, 500 ms
   "2080SP241U01.FP_PARM.AI2_Max" : Real AT %DB4303.DBD166, 500 ms
   "2080SP241U01.FP_PARM.AI2_Min" : Real AT %DB4303.DBD170, 500 ms
   "2080SP241U01.FP_PARM.AI3_Max" : Real AT %DB4303.DBD174, 500 ms
   "2080SP241U01.FP_PARM.AI3_Min" : Real AT %DB4303.DBD178, 500 ms
   "2080SP241U01.FP_PARM.AO1a_Max" : Real AT %DB4303.DBD182, 500 ms
   "2080SP241U01.FP_PARM.AO1a_Min" : Real AT %DB4303.DBD186, 500 ms
   "2080SP241U01.FP_PARM.AO1b_Max" : Real AT %DB4303.DBD206, 500 ms
   "2080SP241U01.FP_PARM.AO1b_Min" : Real AT %DB4303.DBD210, 500 ms
   "2080SP241U01.FP_PARM.AO2a_Max" : Real AT %DB4303.DBD190, 500 ms
   "2080SP241U01.FP_PARM.AO2a_Min" : Real AT %DB4303.DBD194, 500 ms
   "2080SP241U01.FP_PARM.AO2b_Max" : Real AT %DB4303.DBD214, 500 ms
   "2080SP241U01.FP_PARM.AO2b_Min" : Real AT %DB4303.DBD218, 500 ms
   "2080SP241U01.FP_PARM.AO3a_Max" : Real AT %DB4303.DBD198, 500 ms
   "2080SP241U01.FP_PARM.AO3a_Min" : Real AT %DB4303.DBD202, 500 ms
   "2080SP241U01.FP_PARM.AO3b_Max" : Real AT %DB4303.DBD222, 500 ms
   "2080SP241U01.FP_PARM.AO3b_Min" : Real AT %DB4303.DBD226, 500 ms
   "2080SP241U01.FP_PARM.ChangeDir_Acc" : Int AT %DB4303.DBW138, 500 ms
   "2080SP241U01.FP_PARM.ChangeDir_Pre" : Int AT %DB4303.DBW136, 500 ms
   "2080SP241U01.FP_PARM.DelayStart_Acc" : Int AT %DB4303.DBW114, 500 ms
   "2080SP241U01.FP_PARM.DelayStart_Pre" : Int AT %DB4303.DBW112, 500 ms
   "2080SP241U01.FP_PARM.DelayStop_Acc" : Int AT %DB4303.DBW118, 500 ms
   "2080SP241U01.FP_PARM.DelayStop_Pre" : Int AT %DB4303.DBW116, 500 ms
   "2080SP241U01.FP_PARM.INTL" : Bool AT %DB4303.DBX230.0, 500 ms
   "2080SP241U01.FP_PARM.INTL_SEQ_STP" : Bool AT %DB4303.DBX230.3, 500 ms
   "2080SP241U01.FP_PARM.INTL_SEQ_STR1" : Bool AT %DB4303.DBX230.1, 500 ms
   "2080SP241U01.FP_PARM.INTL_SEQ_STR2" : Bool AT %DB4303.DBX230.2, 500 ms
   "2080SP241U01.FP_PARM.LeaveFS_Acc" : Int AT %DB4303.DBW142, 500 ms
   "2080SP241U01.FP_PARM.LeaveFS_Pre" : Int AT %DB4303.DBW140, 500 ms
   "2080SP241U01.FP_PARM.MD_Freq_PV" : Int AT %DB4303.DBW154, 500 ms
   "2080SP241U01.FP_PARM.MD_Freq_SP" : Int AT %DB4303.DBW152, 500 ms
   "2080SP241U01.FP_PARM.ReachFS_Acc" : Int AT %DB4303.DBW150, 500 ms
   "2080SP241U01.FP_PARM.ReachFS_Pre" : Int AT %DB4303.DBW148, 500 ms
   "2080SP241U01.FP_PARM.ReachLS_Acc" : Int AT %DB4303.DBW146, 500 ms
   "2080SP241U01.FP_PARM.ReachLS_Pre" : Int AT %DB4303.DBW144, 500 ms
   "2080SP241U01.FP_PARM.ReturnMon_Acc" : Int AT %DB4303.DBW122, 500 ms
   "2080SP241U01.FP_PARM.ReturnMon_Pre" : Int AT %DB4303.DBW120, 500 ms
   "2080SP241U01.FP_PARM.RunDelay1_Acc" : Int AT %DB4303.DBW106, 500 ms
   "2080SP241U01.FP_PARM.RunDelay1_Pre" : Int AT %DB4303.DBW104, 500 ms
   "2080SP241U01.FP_PARM.RunDelay2_Acc" : Int AT %DB4303.DBW110, 500 ms
   "2080SP241U01.FP_PARM.RunDelay2_Pre" : Int AT %DB4303.DBW108, 500 ms
   "2080SP241U01.FP_PARM.SpeedMonOffDelay_Acc" : Int AT %DB4303.DBW130, 500 ms
   "2080SP241U01.FP_PARM.SpeedMonOffDelay_Pre" : Int AT %DB4303.DBW128, 500 ms
   "2080SP241U01.FP_PARM.SpeedMonOnDelay_Acc" : Int AT %DB4303.DBW126, 500 ms
   "2080SP241U01.FP_PARM.SpeedMonOnDelay_Pre" : Int AT %DB4303.DBW124, 500 ms
   "2080SP241U01.FP_PARM.SpeedMonTrigDelay_Acc" : Int AT %DB4303.DBW134, 500 ms
   "2080SP241U01.FP_PARM.SpeedMonTrigDelay_Pre" : Int AT %DB4303.DBW132, 500 ms
   "2080SP241U01.FP_PARM.StartWarn_Acc" : Int AT %DB4303.DBW102, 500 ms
   "2080SP241U01.FP_PARM.StartWarn_Pre" : Int AT %DB4303.DBW100, 500 ms
   "2080SP241U01.FP_PARM.StopReason" : Int AT %DB4303.DBW156, 500 ms
   "2080SP241U01.FP_SEL.INCH_Loc" : Bool AT %DB4303.DBX87.7, 500 ms
   "2080SP241U01.FP_SEL.INCH_Man" : Bool AT %DB4303.DBX87.6, 500 ms
   "2080SP241U01.FP_SEL.MD" : Bool AT %DB4303.DBX86.0, 500 ms
   "2080SP241U01.FP_SEL.MD_Maintain" : Bool AT %DB4303.DBX86.3, 500 ms
   "2080SP241U01.FP_SEL.MD_OnOff" : Bool AT %DB4303.DBX86.2, 500 ms
   "2080SP241U01.FP_SEL.MD_Puls" : Bool AT %DB4303.DBX86.1, 500 ms
   "2080SP241U01.FP_SEL.MotorStarter" : Bool AT %DB4303.DBX87.3, 500 ms
   "2080SP241U01.FP_SEL.OutOfSevice" : Bool AT %DB4303.DBX88.0, 500 ms
   "2080SP241U01.FP_SEL.ParentCollection" : Bool AT %DB4303.DBX87.5, 500 ms
   "2080SP241U01.FP_SEL.ParentSupress" : Bool AT %DB4303.DBX87.4, 500 ms
   "2080SP241U01.FP_SEL.STW_AutoStart" : Bool AT %DB4303.DBX86.4, 500 ms
   "2080SP241U01.FP_SEL.STW_Local" : Bool AT %DB4303.DBX86.5, 500 ms
   "2080SP241U01.FP_SEL.STW_Manual" : Bool AT %DB4303.DBX86.6, 500 ms
   "2080SP241U01.FP_SEL.STW_Single" : Bool AT %DB4303.DBX86.7, 500 ms
   "2080SP241U01.FP_SEL.Type_Bimotor" : Bool AT %DB4303.DBX87.1, 500 ms
   "2080SP241U01.FP_SEL.Type_Indication" : Bool AT %DB4303.DBX87.2, 500 ms
   "2080SP241U01.FP_SEL.Type_Unimotor" : Bool AT %DB4303.DBX87.0, 500 ms
   "2080SP241U01.FP_SEL.WarningDrive" : Bool AT %DB4303.DBX88.1, 500 ms
   "2080SP241U01.FP_SHOW.ACK" : Bool AT %DB4303.DBX97.5, 500 ms
   "2080SP241U01.FP_SHOW.AI1" : Bool AT %DB4303.DBX95.0, 500 ms
   "2080SP241U01.FP_SHOW.AI2" : Bool AT %DB4303.DBX95.1, 500 ms
   "2080SP241U01.FP_SHOW.AI3" : Bool AT %DB4303.DBX95.2, 500 ms
   "2080SP241U01.FP_SHOW.ASTR" : Bool AT %DB4303.DBX99.2, 500 ms
   "2080SP241U01.FP_SHOW.B1" : Byte AT %DB4303.DBB95, 500 ms
   "2080SP241U01.FP_SHOW.B2" : Byte AT %DB4303.DBB96, 500 ms
   "2080SP241U01.FP_SHOW.B3" : Byte AT %DB4303.DBB97, 500 ms
   "2080SP241U01.FP_SHOW.B4" : Byte AT %DB4303.DBB98, 500 ms
   "2080SP241U01.FP_SHOW.BUSF" : Bool AT %DB4303.DBX97.2, 500 ms
   "2080SP241U01.FP_SHOW.ChangeDir" : Bool AT %DB4303.DBX99.0, 500 ms
   "2080SP241U01.FP_SHOW.CON2" : Bool AT %DB4303.DBX98.2, 500 ms
   "2080SP241U01.FP_SHOW.DelayRun2" : Bool AT %DB4303.DBX98.7, 500 ms
   "2080SP241U01.FP_SHOW.DOPR" : Bool AT %DB4303.DBX97.3, 500 ms
   "2080SP241U01.FP_SHOW.DRDY" : Bool AT %DB4303.DBX96.4, 500 ms
   "2080SP241U01.FP_SHOW.DTEST" : Bool AT %DB4303.DBX97.4, 500 ms
   "2080SP241U01.FP_SHOW.EARTH" : Bool AT %DB4303.DBX96.6, 500 ms
   "2080SP241U01.FP_SHOW.ES" : Bool AT %DB4303.DBX96.2, 500 ms
   "2080SP241U01.FP_SHOW.GFA" : Bool AT %DB4303.DBX97.0, 500 ms
   "2080SP241U01.FP_SHOW.GWA" : Bool AT %DB4303.DBX97.1, 500 ms
   "2080SP241U01.FP_SHOW.LSTP" : Bool AT %DB4303.DBX95.7, 500 ms
   "2080SP241U01.FP_SHOW.LSTR1" : Bool AT %DB4303.DBX97.6, 500 ms
   "2080SP241U01.FP_SHOW.LSTR2" : Bool AT %DB4303.DBX97.7, 500 ms
   "2080SP241U01.FP_SHOW.MCC" : Bool AT %DB4303.DBX95.4, 500 ms
   "2080SP241U01.FP_SHOW.MD" : Bool AT %DB4303.DBX98.6, 500 ms
   "2080SP241U01.FP_SHOW.OVL" : Bool AT %DB4303.DBX95.6, 500 ms
   "2080SP241U01.FP_SHOW.PB_Auto" : Bool AT %DB4303.DBX94.0, 500 ms
   "2080SP241U01.FP_SHOW.PB_Local" : Bool AT %DB4303.DBX94.1, 500 ms
   "2080SP241U01.FP_SHOW.PB_Manual" : Bool AT %DB4303.DBX94.2, 500 ms
   "2080SP241U01.FP_SHOW.PB_QStop" : Bool AT %DB4303.DBX94.7, 500 ms
   "2080SP241U01.FP_SHOW.PB_Reset" : Bool AT %DB4303.DBX99.1, 500 ms
   "2080SP241U01.FP_SHOW.PB_Start1" : Bool AT %DB4303.DBX94.3, 500 ms
   "2080SP241U01.FP_SHOW.PB_Start2" : Bool AT %DB4303.DBX94.4, 500 ms
   "2080SP241U01.FP_SHOW.PB_Stop" : Bool AT %DB4303.DBX94.5, 500 ms
   "2080SP241U01.FP_SHOW.PB_Test" : Bool AT %DB4303.DBX94.6, 500 ms
   "2080SP241U01.FP_SHOW.RD2" : Bool AT %DB4303.DBX98.3, 500 ms
   "2080SP241U01.FP_SHOW.RDY" : Bool AT %DB4303.DBX95.5, 500 ms
   "2080SP241U01.FP_SHOW.REM" : Bool AT %DB4303.DBX96.0, 500 ms
   "2080SP241U01.FP_SHOW.RET2" : Bool AT %DB4303.DBX98.0, 500 ms
   "2080SP241U01.FP_SHOW.RUN2" : Bool AT %DB4303.DBX98.1, 500 ms
   "2080SP241U01.FP_SHOW.SFS" : Bool AT %DB4303.DBX98.4, 500 ms
   "2080SP241U01.FP_SHOW.SLS" : Bool AT %DB4303.DBX98.5, 500 ms
   "2080SP241U01.FP_SHOW.SP" : Bool AT %DB4303.DBX95.3, 500 ms
   "2080SP241U01.FP_SHOW.SSW" : Bool AT %DB4303.DBX96.1, 500 ms
   "2080SP241U01.FP_SHOW.STALL" : Bool AT %DB4303.DBX96.5, 500 ms
   "2080SP241U01.FP_SHOW.TFA" : Bool AT %DB4303.DBX96.3, 500 ms
   "2080SP241U01.FP_SHOW.UBAL" : Bool AT %DB4303.DBX96.7, 500 ms
   "2080SP241U01.ModePointer" : Int AT %DB4303.DBW496, 500 ms
   "2080SP241U01.MSW" : DWord AT %DB4303.DBD62, 500 ms
   "2080SP241U01.ParentInfo" : TextRef, internal   // Имя родителя для попап окна, вкладка инфо. При експорте из ECS через скрипт заполняется автоматически, если теги копируются в ручную то требуется в ручную задатать свойство Start Value
   "2080SP241U01.SPSET" : Real AT %DB4303.DBD18, 500 ms
   "2080SP241U01.StatusWork" : Int AT %DB4303.DBW494, 500 ms

